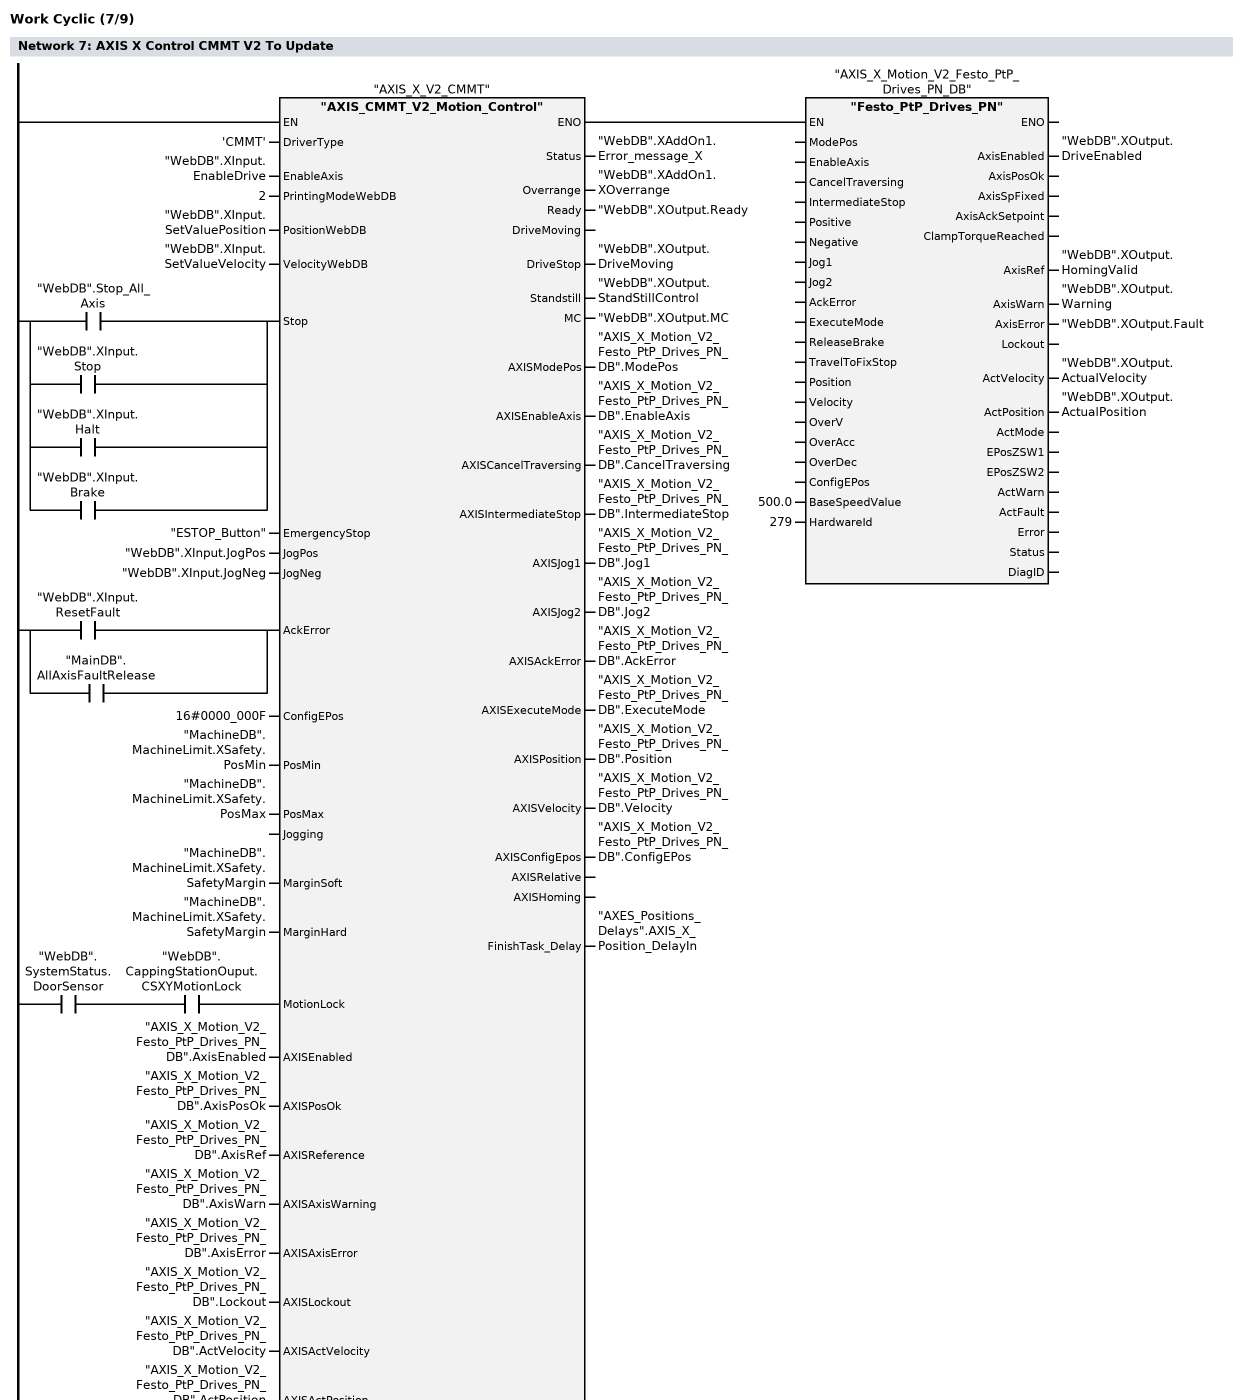
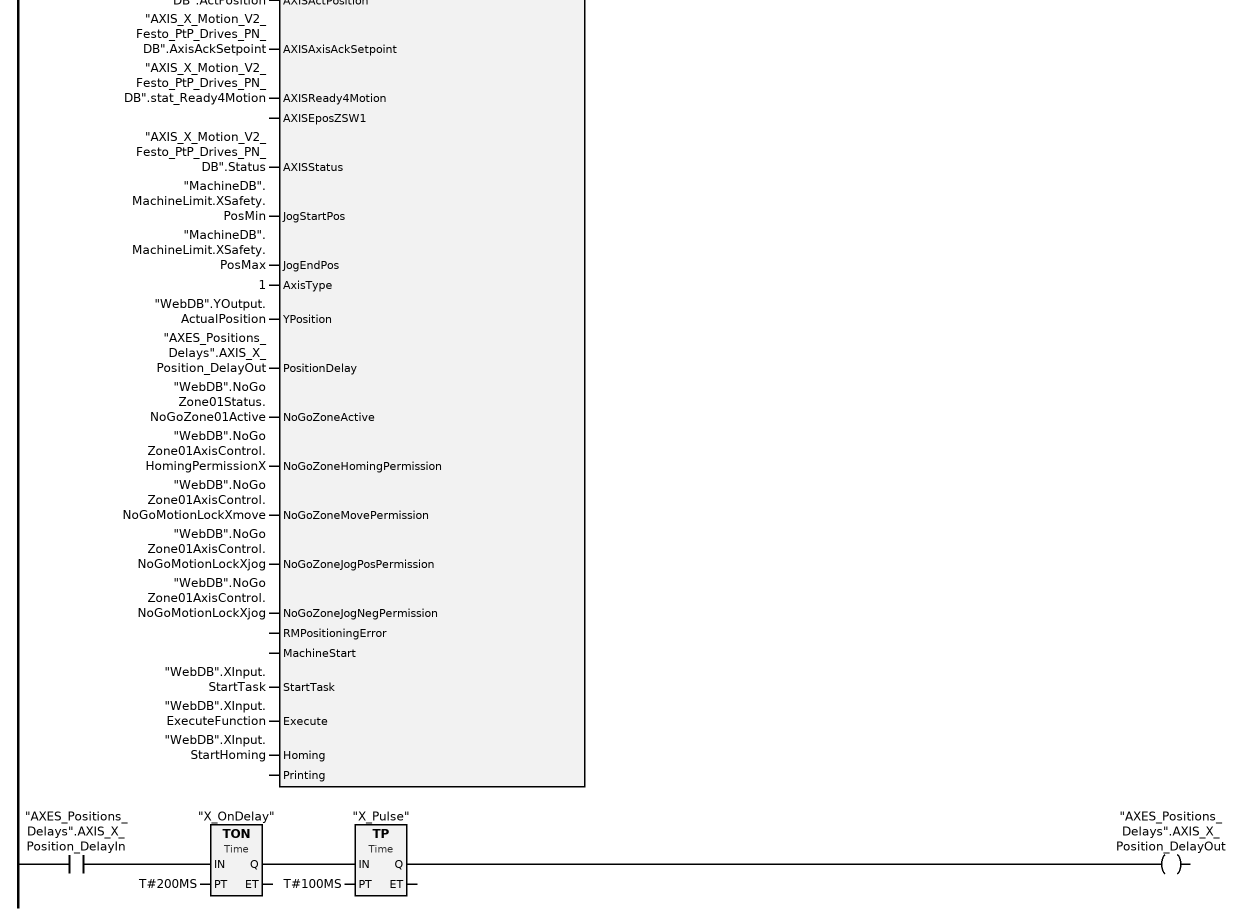
   RUNG wire#powerrail
      "AXIS_X_V2_CMMT"(Stop := wire#w1, AckError := wire#w2, MotionLock := wire#w3, DriverType := 'CMMT', EnableAxis := "WebDB".XInput.EnableDrive, PrintingModeWebDB := 2, PositionWebDB := "WebDB".XInput.SetValuePosition, VelocityWebDB := "WebDB".XInput.SetValueVelocity, EmergencyStop := "ESTOP_Button", JogPos := "WebDB".XInput.JogPos, JogNeg := "WebDB".XInput.JogNeg, ConfigEPos := 16#0000_000F, PosMin := "MachineDB".MachineLimit.XSafety.PosMin, PosMax := "MachineDB".MachineLimit.XSafety.PosMax, Jogging :=, MarginSoft := "MachineDB".MachineLimit.XSafety.SafetyMargin, MarginHard := "MachineDB".MachineLimit.XSafety.SafetyMargin, AXISEnabled := "AXIS_X_Motion_V2_Festo_PtP_Drives_PN_DB".AxisEnabled, AXISPosOk := "AXIS_X_Motion_V2_Festo_PtP_Drives_PN_DB".AxisPosOk, AXISReference := "AXIS_X_Motion_V2_Festo_PtP_Drives_PN_DB".AxisRef, AXISAxisWarning := "AXIS_X_Motion_V2_Festo_PtP_Drives_PN_DB".AxisWarn, AXISAxisError := "AXIS_X_Motion_V2_Festo_PtP_Drives_PN_DB".AxisError, AXISLockout := "AXIS_X_Motion_V2_Festo_PtP_Drives_PN_DB".Lockout, AXISActVelocity := "AXIS_X_Motion_V2_Festo_PtP_Drives_PN_DB".ActVelocity, AXISActPosition := "AXIS_X_Motion_V2_Festo_PtP_Drives_PN_DB".ActPosition, AXISAxisAckSetpoint := "AXIS_X_Motion_V2_Festo_PtP_Drives_PN_DB".AxisAckSetpoint, AXISReady4Motion := "AXIS_X_Motion_V2_Festo_PtP_Drives_PN_DB".stat_Ready4Motion, AXISEposZSW1 :=, AXISStatus := "AXIS_X_Motion_V2_Festo_PtP_Drives_PN_DB".Status, JogStartPos := "MachineDB".MachineLimit.XSafety.PosMin, JogEndPos := "MachineDB".MachineLimit.XSafety.PosMax, AxisType := 1, YPosition := "WebDB".YOutput.ActualPosition, PositionDelay := "AXES_Positions_Delays".AXIS_X_Position_DelayOut, NoGoZoneActive := "WebDB".NoGoZone01Status.NoGoZone01Active, NoGoZoneHomingPermission := "WebDB".NoGoZone01AxisControl.HomingPermissionX, NoGoZoneMovePermission := "WebDB".NoGoZone01AxisControl.NoGoMotionLockXmove, NoGoZoneJogPosPermission := "WebDB".NoGoZone01AxisControl.NoGoMotionLockXjog, NoGoZoneJogNegPermission := "WebDB".NoGoZone01AxisControl.NoGoMotionLockXjog, RMPositioningError :=, MachineStart :=, StartTask := "WebDB".XInput.StartTask, Execute := "WebDB".XInput.ExecuteFunction, Homing := "WebDB".XInput.StartHoming, Printing :=, Status => "WebDB".XAddOn1.Error_message_X, Overrange => "WebDB".XAddOn1.XOverrange, Ready => "WebDB".XOutput.Ready, DriveMoving =>, DriveStop => "WebDB".XOutput.DriveMoving, Standstill => "WebDB".XOutput.StandStillControl, MC => "WebDB".XOutput.MC, AXISModePos => "AXIS_X_Motion_V2_Festo_PtP_Drives_PN_DB".ModePos, AXISEnableAxis => "AXIS_X_Motion_V2_Festo_PtP_Drives_PN_DB".EnableAxis, AXISCancelTraversing => "AXIS_X_Motion_V2_Festo_PtP_Drives_PN_DB".CancelTraversing, AXISIntermediateStop => "AXIS_X_Motion_V2_Festo_PtP_Drives_PN_DB".IntermediateStop, AXISJog1 => "AXIS_X_Motion_V2_Festo_PtP_Drives_PN_DB".Jog1, AXISJog2 => "AXIS_X_Motion_V2_Festo_PtP_Drives_PN_DB".Jog2, AXISAckError => "AXIS_X_Motion_V2_Festo_PtP_Drives_PN_DB".AckError, AXISExecuteMode => "AXIS_X_Motion_V2_Festo_PtP_Drives_PN_DB".ExecuteMode, AXISPosition => "AXIS_X_Motion_V2_Festo_PtP_Drives_PN_DB".Position, AXISVelocity => "AXIS_X_Motion_V2_Festo_PtP_Drives_PN_DB".Velocity, AXISConfigEpos => "AXIS_X_Motion_V2_Festo_PtP_Drives_PN_DB".ConfigEPos, AXISRelative =>, AXISHoming =>, FinishTask_Delay => "AXES_Positions_Delays".AXIS_X_Position_DelayIn)
      "AXIS_X_Motion_V2_Festo_PtP_Drives_PN_DB"(ModePos :=, EnableAxis :=, CancelTraversing :=, IntermediateStop :=, Positive :=, Negative :=, Jog1 :=, Jog2 :=, AckError :=, ExecuteMode :=, ReleaseBrake :=, TravelToFixStop :=, Position :=, Velocity :=, OverV :=, OverAcc :=, OverDec :=, ConfigEPos :=, BaseSpeedValue := 500.0, HardwareId := 279, AxisEnabled => "WebDB".XOutput.DriveEnabled, AxisPosOk =>, AxisSpFixed =>, AxisAckSetpoint =>, ClampTorqueReached =>, AxisRef => "WebDB".XOutput.HomingValid, AxisWarn => "WebDB".XOutput.Warning, AxisError => "WebDB".XOutput.Fault, Lockout =>, ActVelocity => "WebDB".XOutput.ActualVelocity, ActPosition => "WebDB".XOutput.ActualPosition, ActMode =>, EPosZSW1 =>, EPosZSW2 =>, ActWarn =>, ActFault =>, Error =>, Status =>, DiagID =>)
   END_RUNG
   RUNG wire#powerrail
      Contact( "WebDB".Stop_All_Axis )
   END_RUNG wire#w1
   RUNG wire#powerrail
      Contact( "WebDB".XInput.Stop )
   END_RUNG wire#w1
   RUNG wire#powerrail
      Contact( "WebDB".XInput.Halt )
   END_RUNG wire#w1
   RUNG wire#powerrail
      Contact( "WebDB".XInput.Brake )
   END_RUNG wire#w1
   RUNG wire#powerrail
      Contact( "WebDB".XInput.ResetFault )
   END_RUNG wire#w2
   RUNG wire#powerrail
      Contact( "MainDB".AllAxisFaultRelease )
   END_RUNG wire#w2
   RUNG wire#powerrail
      Contact( "WebDB".SystemStatus.DoorSensor )
      Contact( "WebDB".CappingStationOuput.CSXYMotionLock )
   END_RUNG wire#w3
   RUNG wire#powerrail
      Contact( "AXES_Positions_Delays".AXIS_X_Position_DelayIn )
      { S7_Templates := "time_type := Time" } "X_OnDelay".TON(pt := T#200MS, et =>)
      { S7_Templates := "time_type := Time" } "X_Pulse".TP(pt := T#100MS, et =>)
      Coil( "AXES_Positions_Delays".AXIS_X_Position_DelayOut )
   END_RUNG
   // the same network as SCL:
   "AXIS_X_V2_CMMT"(DriverType := 'CMMT',   // "AXIS_CMMT_V2_Motion_Control"
                    EnableAxis := "WebDB".XInput.EnableDrive,
                    PrintingModeWebDB := 2,
                    PositionWebDB := "WebDB".XInput.SetValuePosition,
                    VelocityWebDB := "WebDB".XInput.SetValueVelocity,
                    Stop := "WebDB".Stop_All_Axis OR "WebDB".XInput.Stop OR "WebDB".XInput.Halt OR "WebDB".XInput.Brake,
                    EmergencyStop := "ESTOP_Button",
                    JogPos := "WebDB".XInput.JogPos,
                    JogNeg := "WebDB".XInput.JogNeg,
                    AckError := "WebDB".XInput.ResetFault OR "MainDB".AllAxisFaultRelease,
                    ConfigEPos := 16#0000_000F,
                    PosMin := "MachineDB".MachineLimit.XSafety.PosMin,
                    PosMax := "MachineDB".MachineLimit.XSafety.PosMax,
                    MarginSoft := "MachineDB".MachineLimit.XSafety.SafetyMargin,
                    MarginHard := "MachineDB".MachineLimit.XSafety.SafetyMargin,
                    MotionLock := "WebDB".SystemStatus.DoorSensor AND "WebDB".CappingStationOuput.CSXYMotionLock,
                    AXISEnabled := "AXIS_X_Motion_V2_Festo_PtP_Drives_PN_DB".AxisEnabled,
                    AXISPosOk := "AXIS_X_Motion_V2_Festo_PtP_Drives_PN_DB".AxisPosOk,
                    AXISReference := "AXIS_X_Motion_V2_Festo_PtP_Drives_PN_DB".AxisRef,
                    AXISAxisWarning := "AXIS_X_Motion_V2_Festo_PtP_Drives_PN_DB".AxisWarn,
                    AXISAxisError := "AXIS_X_Motion_V2_Festo_PtP_Drives_PN_DB".AxisError,
                    AXISLockout := "AXIS_X_Motion_V2_Festo_PtP_Drives_PN_DB".Lockout,
                    AXISActVelocity := "AXIS_X_Motion_V2_Festo_PtP_Drives_PN_DB".ActVelocity,
                    AXISActPosition := "AXIS_X_Motion_V2_Festo_PtP_Drives_PN_DB".ActPosition,
                    AXISAxisAckSetpoint := "AXIS_X_Motion_V2_Festo_PtP_Drives_PN_DB".AxisAckSetpoint,
                    AXISReady4Motion := "AXIS_X_Motion_V2_Festo_PtP_Drives_PN_DB".stat_Ready4Motion,
                    AXISStatus := "AXIS_X_Motion_V2_Festo_PtP_Drives_PN_DB".Status,
                    JogStartPos := "MachineDB".MachineLimit.XSafety.PosMin,
                    JogEndPos := "MachineDB".MachineLimit.XSafety.PosMax,
                    AxisType := 1,
                    YPosition := "WebDB".YOutput.ActualPosition,
                    PositionDelay := "AXES_Positions_Delays".AXIS_X_Position_DelayOut,
                    NoGoZoneActive := "WebDB".NoGoZone01Status.NoGoZone01Active,
                    NoGoZoneHomingPermission := "WebDB".NoGoZone01AxisControl.HomingPermissionX,
                    NoGoZoneMovePermission := "WebDB".NoGoZone01AxisControl.NoGoMotionLockXmove,
                    NoGoZoneJogPosPermission := "WebDB".NoGoZone01AxisControl.NoGoMotionLockXjog,
                    NoGoZoneJogNegPermission := "WebDB".NoGoZone01AxisControl.NoGoMotionLockXjog,
                    StartTask := "WebDB".XInput.StartTask,
                    Execute := "WebDB".XInput.ExecuteFunction,
                    Homing := "WebDB".XInput.StartHoming,
                    Status => "WebDB".XAddOn1.Error_message_X,
                    Overrange => "WebDB".XAddOn1.XOverrange,
                    Ready => "WebDB".XOutput.Ready,
                    DriveStop => "WebDB".XOutput.DriveMoving,
                    Standstill => "WebDB".XOutput.StandStillControl,
                    MC => "WebDB".XOutput.MC,
                    AXISModePos => "AXIS_X_Motion_V2_Festo_PtP_Drives_PN_DB".ModePos,
                    AXISEnableAxis => "AXIS_X_Motion_V2_Festo_PtP_Drives_PN_DB".EnableAxis,
                    AXISCancelTraversing => "AXIS_X_Motion_V2_Festo_PtP_Drives_PN_DB".CancelTraversing,
                    AXISIntermediateStop => "AXIS_X_Motion_V2_Festo_PtP_Drives_PN_DB".IntermediateStop,
                    AXISJog1 => "AXIS_X_Motion_V2_Festo_PtP_Drives_PN_DB".Jog1,
                    AXISJog2 => "AXIS_X_Motion_V2_Festo_PtP_Drives_PN_DB".Jog2,
                    AXISAckError => "AXIS_X_Motion_V2_Festo_PtP_Drives_PN_DB".AckError,
                    AXISExecuteMode => "AXIS_X_Motion_V2_Festo_PtP_Drives_PN_DB".ExecuteMode,
                    AXISPosition => "AXIS_X_Motion_V2_Festo_PtP_Drives_PN_DB".Position,
                    AXISVelocity => "AXIS_X_Motion_V2_Festo_PtP_Drives_PN_DB".Velocity,
                    AXISConfigEpos => "AXIS_X_Motion_V2_Festo_PtP_Drives_PN_DB".ConfigEPos,
                    FinishTask_Delay => "AXES_Positions_Delays".AXIS_X_Position_DelayIn,
                    ENO => #_w1);
   IF #_w1 THEN
       "AXIS_X_Motion_V2_Festo_PtP_Drives_PN_DB"(BaseSpeedValue := 500.0,   // "Festo_PtP_Drives_PN"
                               HardwareId := 279,
                               AxisEnabled => "WebDB".XOutput.DriveEnabled,
                               AxisRef => "WebDB".XOutput.HomingValid,
                               AxisWarn => "WebDB".XOutput.Warning,
                               AxisError => "WebDB".XOutput.Fault,
                               ActVelocity => "WebDB".XOutput.ActualVelocity,
                               ActPosition => "WebDB".XOutput.ActualPosition);
   END_IF;
   "X_OnDelay".TON(IN := "AXES_Positions_Delays".AXIS_X_Position_DelayIn, PT := T#200MS);
   "X_Pulse".TP(IN := "X_OnDelay".Q, PT := T#100MS);
   "AXES_Positions_Delays".AXIS_X_Position_DelayOut := "X_Pulse".Q;
END_REGION

REGION Network 8: AXIS Y Control CMMT V2 To Update
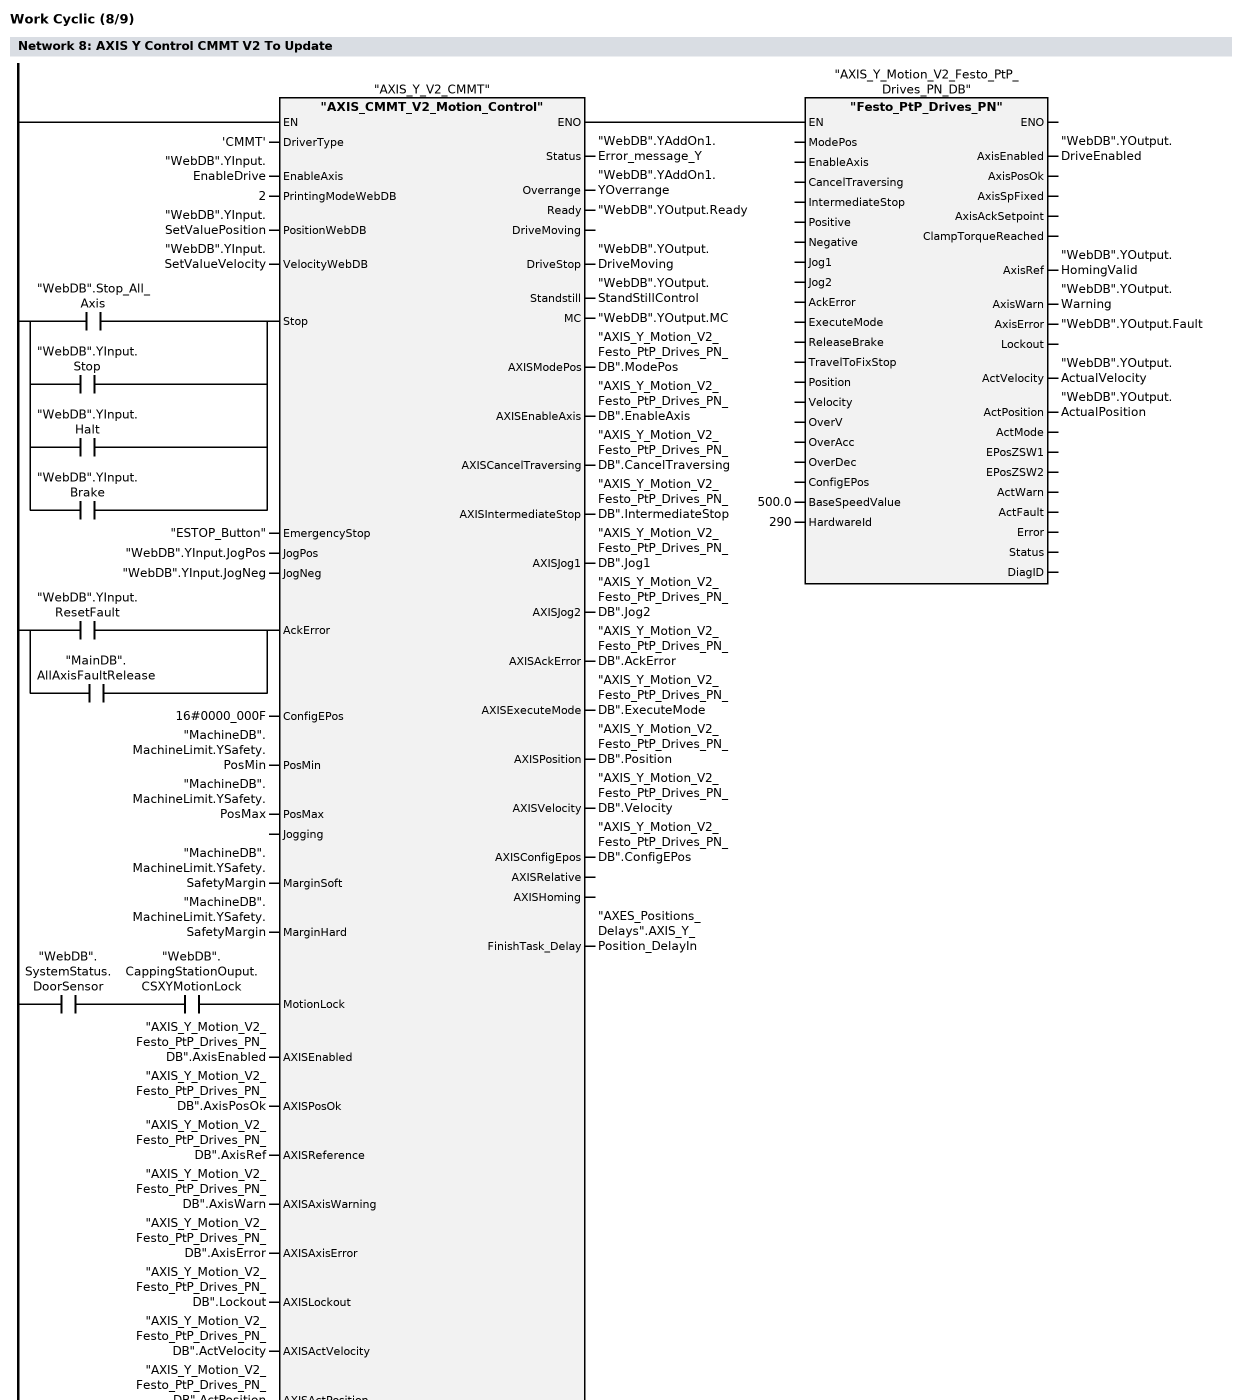
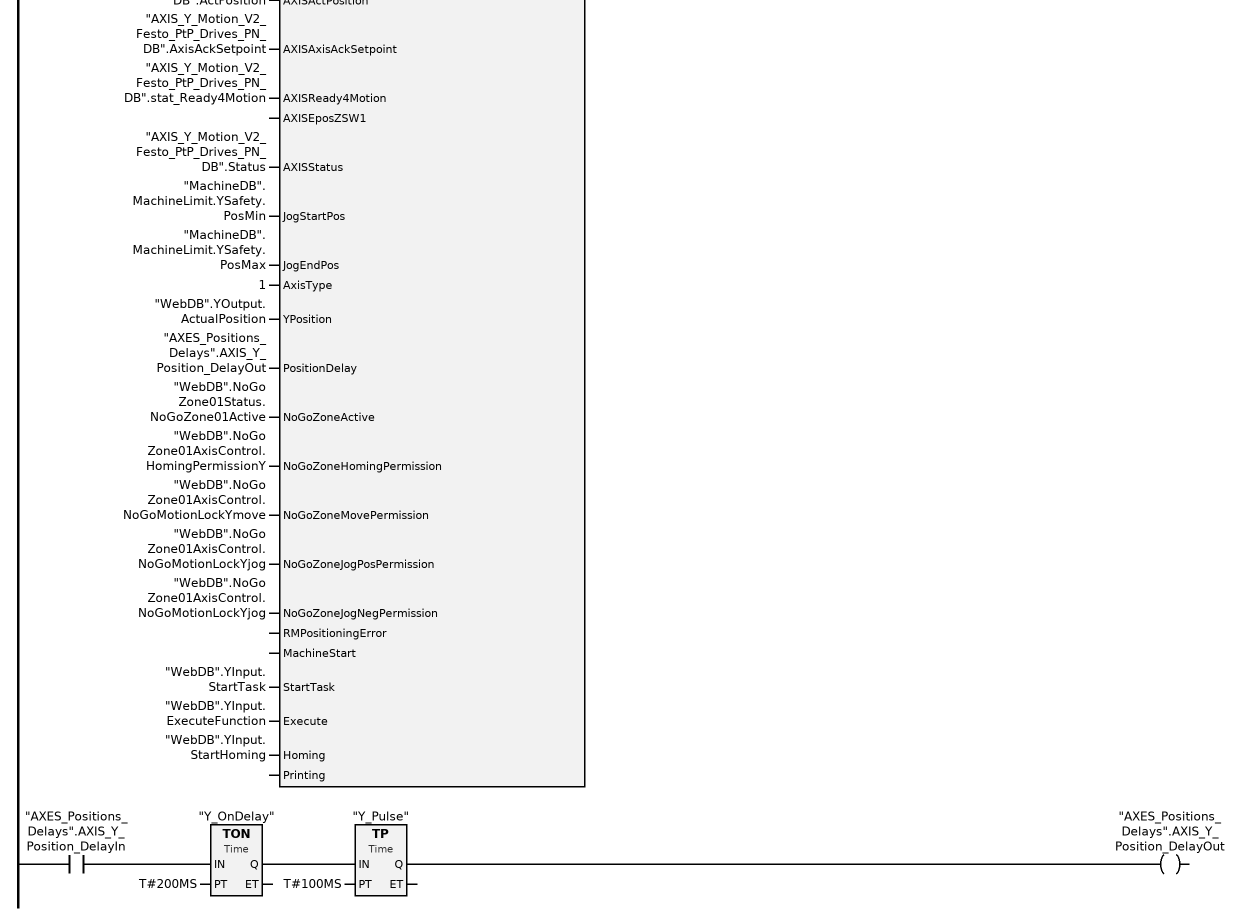
   RUNG wire#powerrail
      "AXIS_Y_V2_CMMT"(Stop := wire#w1, AckError := wire#w2, MotionLock := wire#w3, DriverType := 'CMMT', EnableAxis := "WebDB".YInput.EnableDrive, PrintingModeWebDB := 2, PositionWebDB := "WebDB".YInput.SetValuePosition, VelocityWebDB := "WebDB".YInput.SetValueVelocity, EmergencyStop := "ESTOP_Button", JogPos := "WebDB".YInput.JogPos, JogNeg := "WebDB".YInput.JogNeg, ConfigEPos := 16#0000_000F, PosMin := "MachineDB".MachineLimit.YSafety.PosMin, PosMax := "MachineDB".MachineLimit.YSafety.PosMax, Jogging :=, MarginSoft := "MachineDB".MachineLimit.YSafety.SafetyMargin, MarginHard := "MachineDB".MachineLimit.YSafety.SafetyMargin, AXISEnabled := "AXIS_Y_Motion_V2_Festo_PtP_Drives_PN_DB".AxisEnabled, AXISPosOk := "AXIS_Y_Motion_V2_Festo_PtP_Drives_PN_DB".AxisPosOk, AXISReference := "AXIS_Y_Motion_V2_Festo_PtP_Drives_PN_DB".AxisRef, AXISAxisWarning := "AXIS_Y_Motion_V2_Festo_PtP_Drives_PN_DB".AxisWarn, AXISAxisError := "AXIS_Y_Motion_V2_Festo_PtP_Drives_PN_DB".AxisError, AXISLockout := "AXIS_Y_Motion_V2_Festo_PtP_Drives_PN_DB".Lockout, AXISActVelocity := "AXIS_Y_Motion_V2_Festo_PtP_Drives_PN_DB".ActVelocity, AXISActPosition := "AXIS_Y_Motion_V2_Festo_PtP_Drives_PN_DB".ActPosition, AXISAxisAckSetpoint := "AXIS_Y_Motion_V2_Festo_PtP_Drives_PN_DB".AxisAckSetpoint, AXISReady4Motion := "AXIS_Y_Motion_V2_Festo_PtP_Drives_PN_DB".stat_Ready4Motion, AXISEposZSW1 :=, AXISStatus := "AXIS_Y_Motion_V2_Festo_PtP_Drives_PN_DB".Status, JogStartPos := "MachineDB".MachineLimit.YSafety.PosMin, JogEndPos := "MachineDB".MachineLimit.YSafety.PosMax, AxisType := 1, YPosition := "WebDB".YOutput.ActualPosition, PositionDelay := "AXES_Positions_Delays".AXIS_Y_Position_DelayOut, NoGoZoneActive := "WebDB".NoGoZone01Status.NoGoZone01Active, NoGoZoneHomingPermission := "WebDB".NoGoZone01AxisControl.HomingPermissionY, NoGoZoneMovePermission := "WebDB".NoGoZone01AxisControl.NoGoMotionLockYmove, NoGoZoneJogPosPermission := "WebDB".NoGoZone01AxisControl.NoGoMotionLockYjog, NoGoZoneJogNegPermission := "WebDB".NoGoZone01AxisControl.NoGoMotionLockYjog, RMPositioningError :=, MachineStart :=, StartTask := "WebDB".YInput.StartTask, Execute := "WebDB".YInput.ExecuteFunction, Homing := "WebDB".YInput.StartHoming, Printing :=, Status => "WebDB".YAddOn1.Error_message_Y, Overrange => "WebDB".YAddOn1.YOverrange, Ready => "WebDB".YOutput.Ready, DriveMoving =>, DriveStop => "WebDB".YOutput.DriveMoving, Standstill => "WebDB".YOutput.StandStillControl, MC => "WebDB".YOutput.MC, AXISModePos => "AXIS_Y_Motion_V2_Festo_PtP_Drives_PN_DB".ModePos, AXISEnableAxis => "AXIS_Y_Motion_V2_Festo_PtP_Drives_PN_DB".EnableAxis, AXISCancelTraversing => "AXIS_Y_Motion_V2_Festo_PtP_Drives_PN_DB".CancelTraversing, AXISIntermediateStop => "AXIS_Y_Motion_V2_Festo_PtP_Drives_PN_DB".IntermediateStop, AXISJog1 => "AXIS_Y_Motion_V2_Festo_PtP_Drives_PN_DB".Jog1, AXISJog2 => "AXIS_Y_Motion_V2_Festo_PtP_Drives_PN_DB".Jog2, AXISAckError => "AXIS_Y_Motion_V2_Festo_PtP_Drives_PN_DB".AckError, AXISExecuteMode => "AXIS_Y_Motion_V2_Festo_PtP_Drives_PN_DB".ExecuteMode, AXISPosition => "AXIS_Y_Motion_V2_Festo_PtP_Drives_PN_DB".Position, AXISVelocity => "AXIS_Y_Motion_V2_Festo_PtP_Drives_PN_DB".Velocity, AXISConfigEpos => "AXIS_Y_Motion_V2_Festo_PtP_Drives_PN_DB".ConfigEPos, AXISRelative =>, AXISHoming =>, FinishTask_Delay => "AXES_Positions_Delays".AXIS_Y_Position_DelayIn)
      "AXIS_Y_Motion_V2_Festo_PtP_Drives_PN_DB"(ModePos :=, EnableAxis :=, CancelTraversing :=, IntermediateStop :=, Positive :=, Negative :=, Jog1 :=, Jog2 :=, AckError :=, ExecuteMode :=, ReleaseBrake :=, TravelToFixStop :=, Position :=, Velocity :=, OverV :=, OverAcc :=, OverDec :=, ConfigEPos :=, BaseSpeedValue := 500.0, HardwareId := 290, AxisEnabled => "WebDB".YOutput.DriveEnabled, AxisPosOk =>, AxisSpFixed =>, AxisAckSetpoint =>, ClampTorqueReached =>, AxisRef => "WebDB".YOutput.HomingValid, AxisWarn => "WebDB".YOutput.Warning, AxisError => "WebDB".YOutput.Fault, Lockout =>, ActVelocity => "WebDB".YOutput.ActualVelocity, ActPosition => "WebDB".YOutput.ActualPosition, ActMode =>, EPosZSW1 =>, EPosZSW2 =>, ActWarn =>, ActFault =>, Error =>, Status =>, DiagID =>)
   END_RUNG
   RUNG wire#powerrail
      Contact( "WebDB".Stop_All_Axis )
   END_RUNG wire#w1
   RUNG wire#powerrail
      Contact( "WebDB".YInput.Stop )
   END_RUNG wire#w1
   RUNG wire#powerrail
      Contact( "WebDB".YInput.Halt )
   END_RUNG wire#w1
   RUNG wire#powerrail
      Contact( "WebDB".YInput.Brake )
   END_RUNG wire#w1
   RUNG wire#powerrail
      Contact( "WebDB".YInput.ResetFault )
   END_RUNG wire#w2
   RUNG wire#powerrail
      Contact( "MainDB".AllAxisFaultRelease )
   END_RUNG wire#w2
   RUNG wire#powerrail
      Contact( "WebDB".SystemStatus.DoorSensor )
      Contact( "WebDB".CappingStationOuput.CSXYMotionLock )
   END_RUNG wire#w3
   RUNG wire#powerrail
      Contact( "AXES_Positions_Delays".AXIS_Y_Position_DelayIn )
      { S7_Templates := "time_type := Time" } "Y_OnDelay".TON(pt := T#200MS, et =>)
      { S7_Templates := "time_type := Time" } "Y_Pulse".TP(pt := T#100MS, et =>)
      Coil( "AXES_Positions_Delays".AXIS_Y_Position_DelayOut )
   END_RUNG
   // the same network as SCL:
   "AXIS_Y_V2_CMMT"(DriverType := 'CMMT',   // "AXIS_CMMT_V2_Motion_Control"
                    EnableAxis := "WebDB".YInput.EnableDrive,
                    PrintingModeWebDB := 2,
                    PositionWebDB := "WebDB".YInput.SetValuePosition,
                    VelocityWebDB := "WebDB".YInput.SetValueVelocity,
                    Stop := "WebDB".Stop_All_Axis OR "WebDB".YInput.Stop OR "WebDB".YInput.Halt OR "WebDB".YInput.Brake,
                    EmergencyStop := "ESTOP_Button",
                    JogPos := "WebDB".YInput.JogPos,
                    JogNeg := "WebDB".YInput.JogNeg,
                    AckError := "WebDB".YInput.ResetFault OR "MainDB".AllAxisFaultRelease,
                    ConfigEPos := 16#0000_000F,
                    PosMin := "MachineDB".MachineLimit.YSafety.PosMin,
                    PosMax := "MachineDB".MachineLimit.YSafety.PosMax,
                    MarginSoft := "MachineDB".MachineLimit.YSafety.SafetyMargin,
                    MarginHard := "MachineDB".MachineLimit.YSafety.SafetyMargin,
                    MotionLock := "WebDB".SystemStatus.DoorSensor AND "WebDB".CappingStationOuput.CSXYMotionLock,
                    AXISEnabled := "AXIS_Y_Motion_V2_Festo_PtP_Drives_PN_DB".AxisEnabled,
                    AXISPosOk := "AXIS_Y_Motion_V2_Festo_PtP_Drives_PN_DB".AxisPosOk,
                    AXISReference := "AXIS_Y_Motion_V2_Festo_PtP_Drives_PN_DB".AxisRef,
                    AXISAxisWarning := "AXIS_Y_Motion_V2_Festo_PtP_Drives_PN_DB".AxisWarn,
                    AXISAxisError := "AXIS_Y_Motion_V2_Festo_PtP_Drives_PN_DB".AxisError,
                    AXISLockout := "AXIS_Y_Motion_V2_Festo_PtP_Drives_PN_DB".Lockout,
                    AXISActVelocity := "AXIS_Y_Motion_V2_Festo_PtP_Drives_PN_DB".ActVelocity,
                    AXISActPosition := "AXIS_Y_Motion_V2_Festo_PtP_Drives_PN_DB".ActPosition,
                    AXISAxisAckSetpoint := "AXIS_Y_Motion_V2_Festo_PtP_Drives_PN_DB".AxisAckSetpoint,
                    AXISReady4Motion := "AXIS_Y_Motion_V2_Festo_PtP_Drives_PN_DB".stat_Ready4Motion,
                    AXISStatus := "AXIS_Y_Motion_V2_Festo_PtP_Drives_PN_DB".Status,
                    JogStartPos := "MachineDB".MachineLimit.YSafety.PosMin,
                    JogEndPos := "MachineDB".MachineLimit.YSafety.PosMax,
                    AxisType := 1,
                    YPosition := "WebDB".YOutput.ActualPosition,
                    PositionDelay := "AXES_Positions_Delays".AXIS_Y_Position_DelayOut,
                    NoGoZoneActive := "WebDB".NoGoZone01Status.NoGoZone01Active,
                    NoGoZoneHomingPermission := "WebDB".NoGoZone01AxisControl.HomingPermissionY,
                    NoGoZoneMovePermission := "WebDB".NoGoZone01AxisControl.NoGoMotionLockYmove,
                    NoGoZoneJogPosPermission := "WebDB".NoGoZone01AxisControl.NoGoMotionLockYjog,
                    NoGoZoneJogNegPermission := "WebDB".NoGoZone01AxisControl.NoGoMotionLockYjog,
                    StartTask := "WebDB".YInput.StartTask,
                    Execute := "WebDB".YInput.ExecuteFunction,
                    Homing := "WebDB".YInput.StartHoming,
                    Status => "WebDB".YAddOn1.Error_message_Y,
                    Overrange => "WebDB".YAddOn1.YOverrange,
                    Ready => "WebDB".YOutput.Ready,
                    DriveStop => "WebDB".YOutput.DriveMoving,
                    Standstill => "WebDB".YOutput.StandStillControl,
                    MC => "WebDB".YOutput.MC,
                    AXISModePos => "AXIS_Y_Motion_V2_Festo_PtP_Drives_PN_DB".ModePos,
                    AXISEnableAxis => "AXIS_Y_Motion_V2_Festo_PtP_Drives_PN_DB".EnableAxis,
                    AXISCancelTraversing => "AXIS_Y_Motion_V2_Festo_PtP_Drives_PN_DB".CancelTraversing,
                    AXISIntermediateStop => "AXIS_Y_Motion_V2_Festo_PtP_Drives_PN_DB".IntermediateStop,
                    AXISJog1 => "AXIS_Y_Motion_V2_Festo_PtP_Drives_PN_DB".Jog1,
                    AXISJog2 => "AXIS_Y_Motion_V2_Festo_PtP_Drives_PN_DB".Jog2,
                    AXISAckError => "AXIS_Y_Motion_V2_Festo_PtP_Drives_PN_DB".AckError,
                    AXISExecuteMode => "AXIS_Y_Motion_V2_Festo_PtP_Drives_PN_DB".ExecuteMode,
                    AXISPosition => "AXIS_Y_Motion_V2_Festo_PtP_Drives_PN_DB".Position,
                    AXISVelocity => "AXIS_Y_Motion_V2_Festo_PtP_Drives_PN_DB".Velocity,
                    AXISConfigEpos => "AXIS_Y_Motion_V2_Festo_PtP_Drives_PN_DB".ConfigEPos,
                    FinishTask_Delay => "AXES_Positions_Delays".AXIS_Y_Position_DelayIn,
                    ENO => #_w1);
   IF #_w1 THEN
       "AXIS_Y_Motion_V2_Festo_PtP_Drives_PN_DB"(BaseSpeedValue := 500.0,   // "Festo_PtP_Drives_PN"
                               HardwareId := 290,
                               AxisEnabled => "WebDB".YOutput.DriveEnabled,
                               AxisRef => "WebDB".YOutput.HomingValid,
                               AxisWarn => "WebDB".YOutput.Warning,
                               AxisError => "WebDB".YOutput.Fault,
                               ActVelocity => "WebDB".YOutput.ActualVelocity,
                               ActPosition => "WebDB".YOutput.ActualPosition);
   END_IF;
   "Y_OnDelay".TON(IN := "AXES_Positions_Delays".AXIS_Y_Position_DelayIn, PT := T#200MS);
   "Y_Pulse".TP(IN := "Y_OnDelay".Q, PT := T#100MS);
   "AXES_Positions_Delays".AXIS_Y_Position_DelayOut := "Y_Pulse".Q;
END_REGION

REGION Network 9: Roller V3
   // The RollerV3 block already writes the roller speed and direction to the technology object. This means that the outputs are no longer needed.
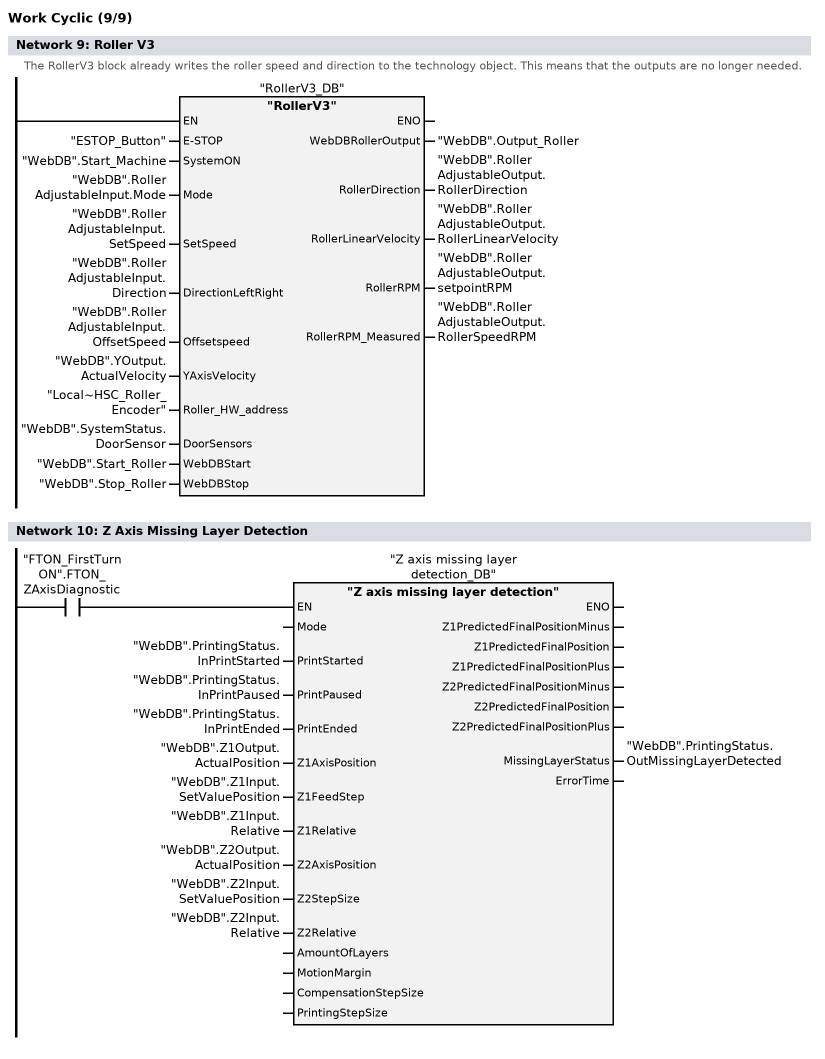
   RUNG wire#powerrail
      "RollerV3_DB"("E-STOP" := "ESTOP_Button", SystemON := "WebDB".Start_Machine, Mode := "WebDB".RollerAdjustableInput.Mode, SetSpeed := "WebDB".RollerAdjustableInput.SetSpeed, DirectionLeftRight := "WebDB".RollerAdjustableInput.Direction, Offsetspeed := "WebDB".RollerAdjustableInput.OffsetSpeed, YAxisVelocity := "WebDB".YOutput.ActualVelocity, Roller_HW_address := "Local~HSC_Roller_Encoder", DoorSensors := "WebDB".SystemStatus.DoorSensor, WebDBStart := "WebDB".Start_Roller, WebDBStop := "WebDB".Stop_Roller, WebDBRollerOutput => "WebDB".Output_Roller, RollerDirection => "WebDB".RollerAdjustableOutput.RollerDirection, RollerLinearVelocity => "WebDB".RollerAdjustableOutput.RollerLinearVelocity, RollerRPM => "WebDB".RollerAdjustableOutput.setpointRPM, RollerRPM_Measured => "WebDB".RollerAdjustableOutput.RollerSpeedRPM)
   END_RUNG
   // the same network as SCL:
   "RollerV3_DB"("E-STOP" := "ESTOP_Button",   // "RollerV3"
                 SystemON := "WebDB".Start_Machine,
                 Mode := "WebDB".RollerAdjustableInput.Mode,
                 SetSpeed := "WebDB".RollerAdjustableInput.SetSpeed,
                 DirectionLeftRight := "WebDB".RollerAdjustableInput.Direction,
                 Offsetspeed := "WebDB".RollerAdjustableInput.OffsetSpeed,
                 YAxisVelocity := "WebDB".YOutput.ActualVelocity,
                 Roller_HW_address := "Local~HSC_Roller_Encoder",
                 DoorSensors := "WebDB".SystemStatus.DoorSensor,
                 WebDBStart := "WebDB".Start_Roller,
                 WebDBStop := "WebDB".Stop_Roller,
                 WebDBRollerOutput => "WebDB".Output_Roller,
                 RollerDirection => "WebDB".RollerAdjustableOutput.RollerDirection,
                 RollerLinearVelocity => "WebDB".RollerAdjustableOutput.RollerLinearVelocity,
                 RollerRPM => "WebDB".RollerAdjustableOutput.setpointRPM,
                 RollerRPM_Measured => "WebDB".RollerAdjustableOutput.RollerSpeedRPM);
END_REGION

REGION Network 10: Z Axis Missing Layer Detection
   RUNG wire#powerrail
      Contact( "FTON_FirstTurnON".FTON_ZAxisDiagnostic )
      "Z axis missing layer detection_DB"(Mode :=, PrintStarted := "WebDB".PrintingStatus.InPrintStarted, PrintPaused := "WebDB".PrintingStatus.InPrintPaused, PrintEnded := "WebDB".PrintingStatus.InPrintEnded, Z1AxisPosition := "WebDB".Z1Output.ActualPosition, Z1FeedStep := "WebDB".Z1Input.SetValuePosition, Z1Relative := "WebDB".Z1Input.Relative, Z2AxisPosition := "WebDB".Z2Output.ActualPosition, Z2StepSize := "WebDB".Z2Input.SetValuePosition, Z2Relative := "WebDB".Z2Input.Relative, AmountOfLayers :=, MotionMargin :=, CompensationStepSize :=, PrintingStepSize :=, Z1PredictedFinalPositionMinus =>, Z1PredictedFinalPosition =>, Z1PredictedFinalPositionPlus =>, Z2PredictedFinalPositionMinus =>, Z2PredictedFinalPosition =>, Z2PredictedFinalPositionPlus =>, MissingLayerStatus => "WebDB".PrintingStatus.OutMissingLayerDetected, ErrorTime =>)
   END_RUNG
   // the same network as SCL:
   IF "FTON_FirstTurnON".FTON_ZAxisDiagnostic THEN
       "Z axis missing layer detection_DB"(PrintStarted := "WebDB".PrintingStatus.InPrintStarted,   // "Z axis missing layer detection"
                               PrintPaused := "WebDB".PrintingStatus.InPrintPaused,
                               PrintEnded := "WebDB".PrintingStatus.InPrintEnded,
                               Z1AxisPosition := "WebDB".Z1Output.ActualPosition,
                               Z1FeedStep := "WebDB".Z1Input.SetValuePosition,
                               Z1Relative := "WebDB".Z1Input.Relative,
                               Z2AxisPosition := "WebDB".Z2Output.ActualPosition,
                               Z2StepSize := "WebDB".Z2Input.SetValuePosition,
                               Z2Relative := "WebDB".Z2Input.Relative,
                               MissingLayerStatus => "WebDB".PrintingStatus.OutMissingLayerDetected);
   END_IF;
END_REGION
END_ORGANIZATION_BLOCK

FUNCTION_BLOCK "AXIS_CMMT_V2_Motion_Control"   // FB22, LAD
TITLE = Description
{ S7_Optimized_Access := 'TRUE' }
VERSION : 0.1
// This is the motion function block used to control all the axes. Due to some differences in the control part for different types of motion and drives, there are additional conditions in some parts of the code.
// 
// Important things to check if the drive is not moving:
// - homing
// - motion lock from add ons (capping station, no go zones)
// - door sensors
// - operation mode
// - communication with the drives (Online access)
   VAR_INPUT
      DriverType : String;   // CMMT; CMMS;
      EnableAxis : Bool;
      PrintingModeWebDB : Int;   // Used while executing the movement
      PositionWebDB : DInt;
      VelocityWebDB : Real;
      Stop : Bool;
      EmergencyStop : Bool;
      JogPos : Bool;
      JogNeg : Bool;
      AckError : Bool;
      ConfigEPos : DWord;
      PosMin : DInt;
      PosMax : DInt;
      Jogging : Bool;
      MarginSoft : DInt;
      MarginHard : DInt;
      MotionLock : Bool;   // Axis will not move is this bool is 0
      AXISEnabled : Bool;
      AXISPosOk : Bool;
      AXISReference : Bool;
      AXISAxisWarning : Bool;
      AXISAxisError : Bool;
      AXISLockout : Bool;
      AXISActVelocity : Real;
      AXISActPosition : DInt;
      AXISAxisAckSetpoint : Bool;
      AXISReady4Motion : Bool;
      AXISEposZSW1 : Word;
      AXISStatus : Word;
      JogStartPos : DInt;   // Limit for jogging
      JogEndPos : DInt;   // Limit for jogging
      AxisType : Int;   // Axis Type: 1 - X; 2 - Y; 3 - Z1; 4 - Z2
      YPosition : DInt;
      PositionDelay : Bool;   // Delay to make it easier to confirm that the motion was finished
      NoGoZoneActive : Bool;   // 1 to activate no go zone
      NoGoZoneHomingPermission : Bool;
      NoGoZoneMovePermission : Bool;
      NoGoZoneJogPosPermission : Bool;
      NoGoZoneJogNegPermission : Bool;
      RMPositioningError : DInt := 5;   // Input Relativer Motion Position Error that we accept
      MachineStart : Bool;
   END_VAR
   VAR_OUTPUT
      Status : Word;
      Overrange : Bool;
      Ready : Bool;
      DriveMoving : Bool;
      DriveStop : Bool;
      Standstill : Bool;
      MC : Bool;
      AXISModePos : Int;
      AXISEnableAxis : Bool;
      AXISCancelTraversing : Bool;
      AXISIntermediateStop : Bool;
      AXISJog1 : Bool;
      AXISJog2 : Bool;
      AXISAckError : Bool;
      AXISExecuteMode : Bool;
      AXISPosition : DInt;
      AXISVelocity : Real;
      AXISConfigEpos : DWord;
      AXISRelative : Bool;
      AXISHoming : Bool;
      FinishTask_Delay : Bool;
   END_VAR
   VAR_IN_OUT
      StartTask : Bool;
      Execute : Bool;
      Homing : Bool;
      Printing : Bool;
   END_VAR
   VAR
      ExecutingMemory : Bool;
      HomingMemory : Bool;
      TaskMemory : Bool;
      ModePos : Int := 4;
      PosOk : Bool;
      Reference : Bool;
      PositionInternal : DInt;
      LockoutInternal : Bool;
      RelativeMode : Bool;   // Mode 1
      AbsoluteMode : Bool;   // Mode 2
      TaskFinished : Bool;
      JoggingXPermission : Bool;
      JoggingYPermission : Bool;
      JoggingPOSZ1Z2Permission : Bool;
      JoggingNEGZ1Z2Permission : Bool;
      JoggingPosMax : DInt;
      JoggingPosMin : DInt;
      JoggingPositionCorrection : DInt := 1500;
      ProfinetDisconnected : Bool;
      PositionStepPlus : DInt;
      CMMT : Bool;
      CMMS : Bool;
      RMStepStartPosition : DInt;   // Relative Motion Step Start Position
      RMPredictedPosition : DInt;   // Relative Motion Predicted Position
      RMFinalPosition : DInt;   // Relative Motion Final Position
      RMLastStepPositionError : DInt;   // Relative Motion Last Step Position Error
      RMStartTaskM01 : Bool;   // Relative Motion Start Task M Positive
      RMStartTaksM02 : Bool;   // Relative Motion Start Task M Negative
      RMStepRangePlus : DInt;
      RMStepRangeMinus : DInt;
      RelativeDirectionInRange : Bool;
   END_VAR
   VAR_TEMP
      RelativeModeHomingM : Bool;
      Jog1_pos : Bool;   // Jog positive direction
      Jog2_neg : Bool;   // Jog negative direction
      Memory1 : Bool;
      Memory2 : Bool;
      PosMinSoft : DInt;
      PosMaxSoft : DInt;
      InternalError : Bool;
      InternalWarning : Bool;
      ExecuteBusy : Bool;
      ExecutingInternal : Bool;
      HomingInternal : Bool;
      TaskInternal : Bool;
      Position_Plus : DInt;
      Position_Minus : DInt;
      TestFinished : Bool;
   END_VAR
   VAR CONSTANT
      Position_Error : DInt := 10;
   END_VAR
   VAR_TEMP   // added for the SCL form of the ladder/FBD networks
      _w1 : Bool;
      _w2 : Bool;
      _w3 : Bool;
   END_VAR
BEGIN

REGION Network 1: Checking driver type
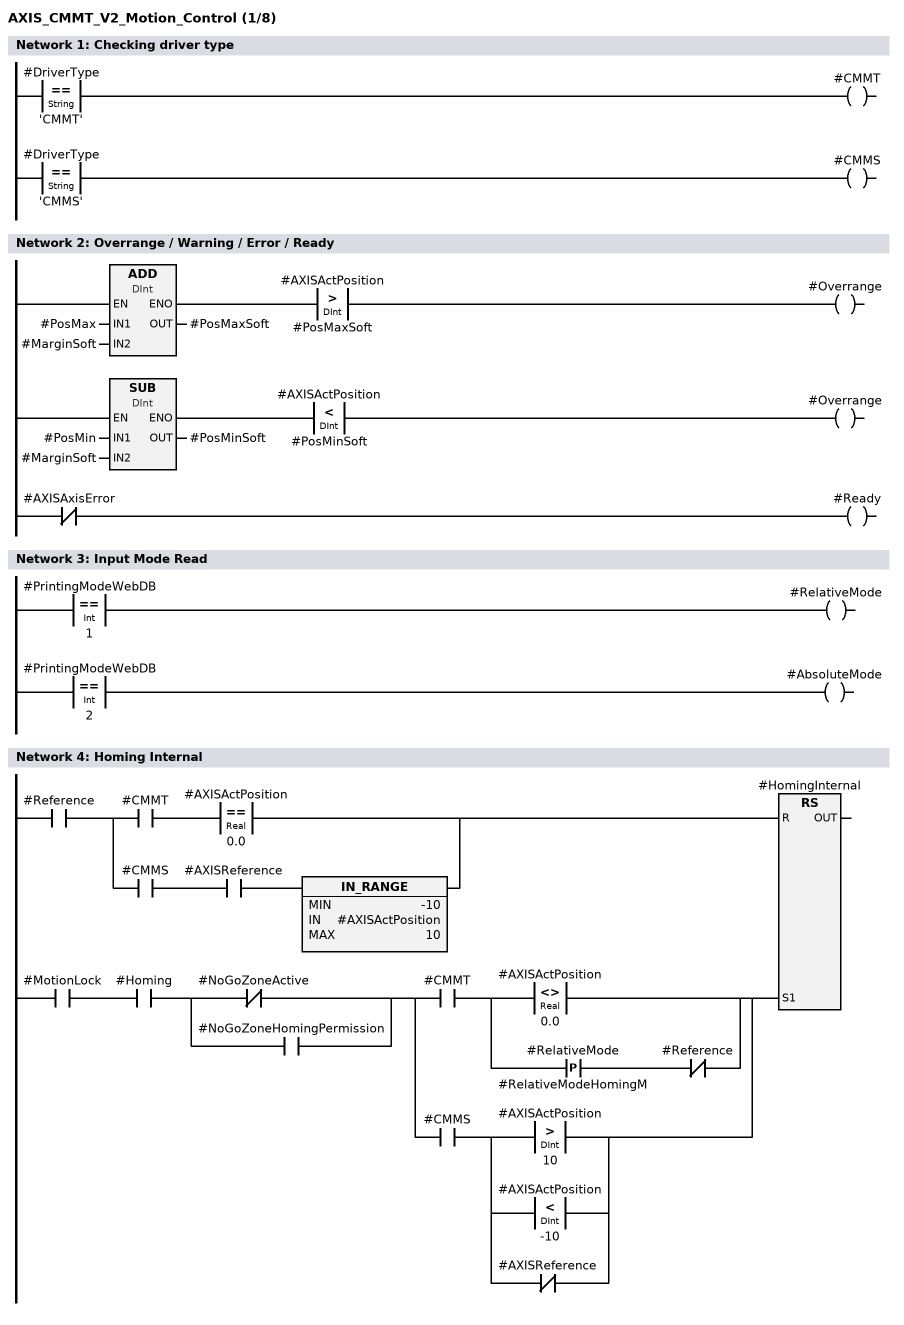
   RUNG wire#powerrail
      { S7_Templates := "SrcType := String" } EQ_Contact(in1 := #DriverType, in2 := 'CMMT')
      Coil( #CMMT )
   END_RUNG
   RUNG wire#powerrail
      { S7_Templates := "SrcType := String" } EQ_Contact(in1 := #DriverType, in2 := 'CMMS')
      Coil( #CMMS )
   END_RUNG
   // the same network as SCL:
   #CMMT := #DriverType = 'CMMT';
   #CMMS := #DriverType = 'CMMS';
END_REGION

REGION Network 2: Overrange / Warning / Error / Ready
   RUNG wire#powerrail
      { S7_Templates := "SrcType := DInt" } Add(in1 := #PosMax, in2 := #MarginSoft, out => #PosMaxSoft)
      { S7_Templates := "SrcType := DInt" } GT_Contact(in1 := #AXISActPosition, in2 := #PosMaxSoft)
      Coil( #Overrange )
   END_RUNG
   RUNG wire#powerrail
      { S7_Templates := "SrcType := DInt" } Sub(in1 := #PosMin, in2 := #MarginSoft, out => #PosMinSoft)
      { S7_Templates := "SrcType := DInt" } LT_Contact(in1 := #AXISActPosition, in2 := #PosMinSoft)
      Coil( #Overrange )
   END_RUNG
   RUNG wire#powerrail
      I_Contact( #AXISAxisError )
      Coil( #Ready )
   END_RUNG
   // the same network as SCL:
   #PosMaxSoft := #PosMax + #MarginSoft;
   #Overrange := #AXISActPosition > #PosMaxSoft;
   #PosMinSoft := #PosMin - #MarginSoft;
   #Overrange := #AXISActPosition < #PosMinSoft;
   #Ready := NOT #AXISAxisError;
END_REGION

REGION Network 3: Input Mode Read
   RUNG wire#powerrail
      { S7_Templates := "SrcType := Int" } EQ_Contact(in1 := #PrintingModeWebDB, in2 := 1)
      Coil( #RelativeMode )
   END_RUNG
   RUNG wire#powerrail
      { S7_Templates := "SrcType := Int" } EQ_Contact(in1 := #PrintingModeWebDB, in2 := 2)
      Coil( #AbsoluteMode )
   END_RUNG
   // the same network as SCL:
   #RelativeMode := #PrintingModeWebDB = 1;
   #AbsoluteMode := #PrintingModeWebDB = 2;
END_REGION

REGION Network 4: Homing Internal
   RUNG wire#powerrail
      Contact( #Reference )
      wire#w1
      Contact( #CMMT )
      { S7_Templates := "SrcType := Real" } EQ_Contact(in1 := #AXISActPosition, in2 := 0.0)
      wire#w2
      S_RS(operand := #HomingInternal, s1 := wire#w7)
   END_RUNG
   RUNG wire#w1
      Contact( #CMMS )
      Contact( #AXISReference )
      { S7_Templates := "SrcType := DInt" } InRange(min := -10, in := #AXISActPosition, max := 10)
   END_RUNG wire#w2
   RUNG wire#powerrail
      Contact( #MotionLock )
      Contact( #Homing )
      wire#w3
      I_Contact( #NoGoZoneActive )
      wire#w4
      Contact( #CMMT )
      wire#w5
      { S7_Templates := "SrcType := Real" } NE_Contact(in1 := #AXISActPosition, in2 := 0.0)
   END_RUNG wire#w7
   RUNG wire#w3
      Contact( #NoGoZoneHomingPermission )
   END_RUNG wire#w4
   RUNG wire#w5
      P_Contact(operand := #RelativeMode, bit := #RelativeModeHomingM)
      I_Contact( #Reference )
   END_RUNG wire#w7
   RUNG wire#w4
      Contact( #CMMS )
      wire#w6
      { S7_Templates := "SrcType := DInt" } GT_Contact(in1 := #AXISActPosition, in2 := 10)
   END_RUNG wire#w7
   RUNG wire#w6
      { S7_Templates := "SrcType := DInt" } LT_Contact(in1 := #AXISActPosition, in2 := -10)
   END_RUNG wire#w7
   RUNG wire#w6
      I_Contact( #AXISReference )
   END_RUNG wire#w7
   // the same network as SCL:
   #_w1 := #MotionLock AND #Homing AND (NOT #NoGoZoneActive OR #NoGoZoneHomingPermission) AND #CMMT AND #RelativeMode AND NOT #RelativeModeHomingM;   // rising edge of #RelativeMode
   #RelativeModeHomingM := #RelativeMode;
   IF #Reference AND ((#CMMT AND (#AXISActPosition = 0.0)) OR (#CMMS AND #AXISReference AND (-10 <= #AXISActPosition) AND (#AXISActPosition <= 10))) THEN
       #HomingInternal := FALSE;   // RS flip-flop
   END_IF;
   IF (#MotionLock AND #Homing AND (NOT #NoGoZoneActive OR #NoGoZoneHomingPermission) AND #CMMT AND (#AXISActPosition <> 0.0)) OR (#_w1 AND NOT #Reference) OR (#MotionLock AND #Homing AND (NOT #NoGoZoneActive OR #NoGoZoneHomingPermission) AND #CMMS AND ((#AXISActPosition > 10) OR (#AXISActPosition < (-10)) OR NOT #AXISReference)) THEN
       #HomingInternal := TRUE;
   END_IF;
END_REGION

REGION Network 5: Status Behavior
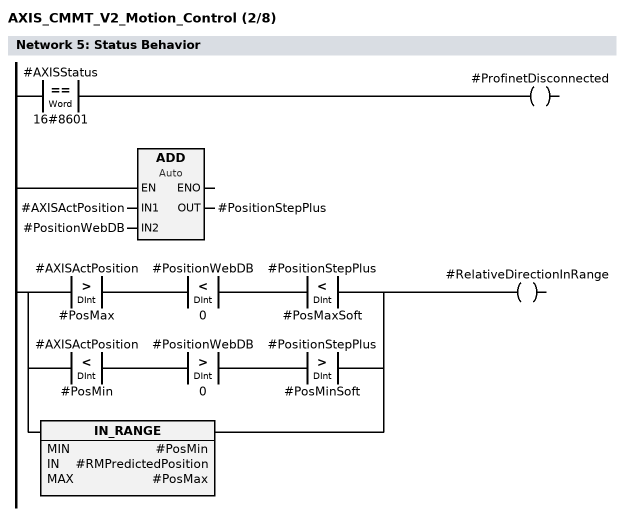
   RUNG wire#powerrail
      { S7_Templates := "SrcType := Word" } EQ_Contact(in1 := #AXISStatus, in2 := 16#8601)
      Coil( #ProfinetDisconnected )
   END_RUNG
   RUNG wire#powerrail
      Add(in1 := #AXISActPosition, in2 := #PositionWebDB, out => #PositionStepPlus)
   END_RUNG
   RUNG wire#powerrail
      { S7_Templates := "SrcType := DInt" } GT_Contact(in1 := #AXISActPosition, in2 := #PosMax)
      { S7_Templates := "SrcType := DInt" } LT_Contact(in1 := #PositionWebDB, in2 := 0)
      { S7_Templates := "SrcType := DInt" } LT_Contact(in1 := #PositionStepPlus, in2 := #PosMaxSoft)
      wire#w1
      Coil( #RelativeDirectionInRange )
   END_RUNG
   RUNG wire#powerrail
      { S7_Templates := "SrcType := DInt" } LT_Contact(in1 := #AXISActPosition, in2 := #PosMin)
      { S7_Templates := "SrcType := DInt" } GT_Contact(in1 := #PositionWebDB, in2 := 0)
      { S7_Templates := "SrcType := DInt" } GT_Contact(in1 := #PositionStepPlus, in2 := #PosMinSoft)
   END_RUNG wire#w1
   RUNG wire#powerrail
      { S7_Templates := "SrcType := DInt" } InRange(min := #PosMin, in := #RMPredictedPosition, max := #PosMax)
   END_RUNG wire#w1
   // the same network as SCL:
   #ProfinetDisconnected := #AXISStatus = 16#8601;
   #PositionStepPlus := #AXISActPosition + #PositionWebDB;
   #RelativeDirectionInRange := ((#AXISActPosition > #PosMax) AND (#PositionWebDB < 0) AND (#PositionStepPlus < #PosMaxSoft)) OR ((#AXISActPosition < #PosMin) AND (#PositionWebDB > 0) AND (#PositionStepPlus > #PosMinSoft)) OR ((#PosMin <= #RMPredictedPosition) AND (#RMPredictedPosition <= #PosMax));
END_REGION

REGION Network 6: Task Internal
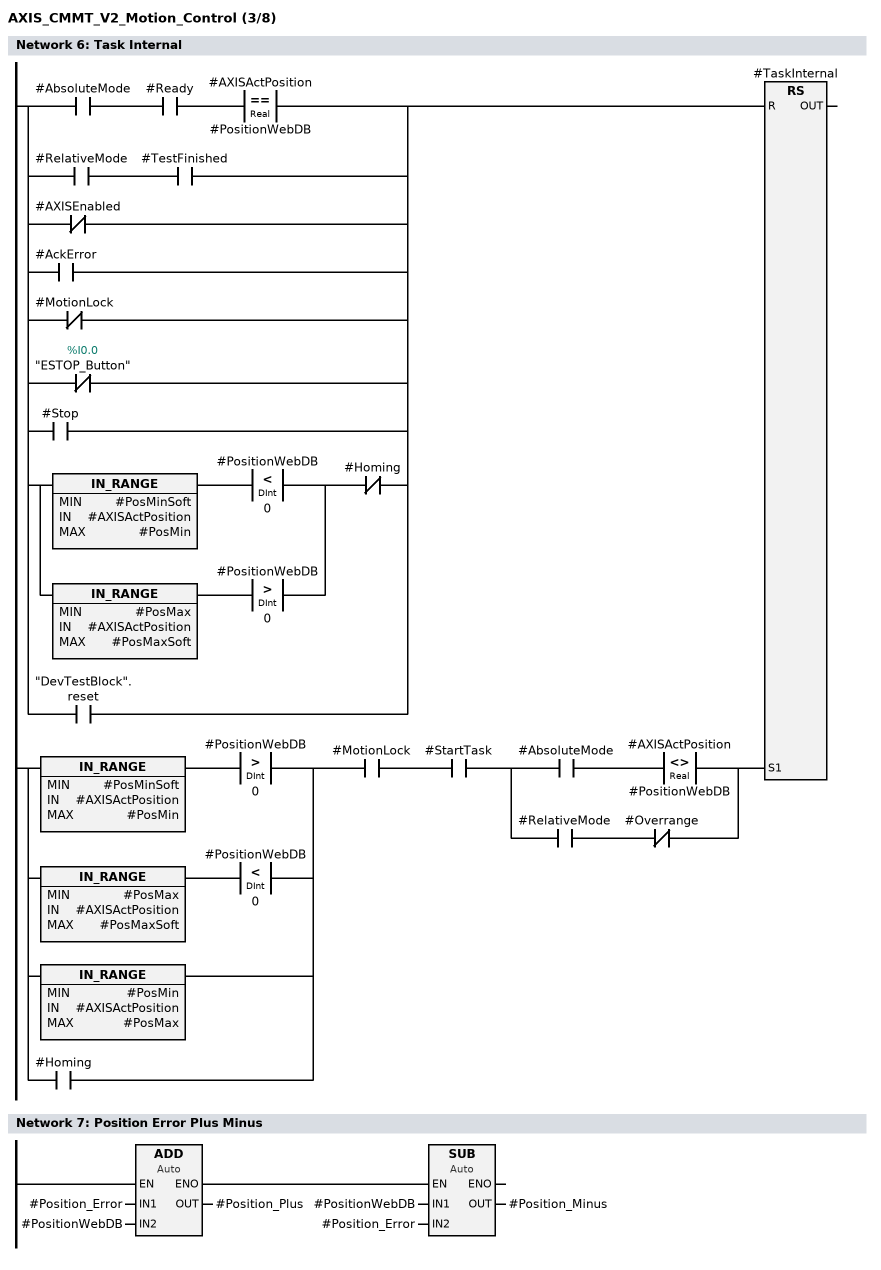
   RUNG wire#powerrail
      Contact( #AbsoluteMode )
      Contact( #Ready )
      { S7_Templates := "SrcType := Real" } EQ_Contact(in1 := #AXISActPosition, in2 := #PositionWebDB)
      wire#w1
      S_RS(operand := #TaskInternal, s1 := wire#w5)
   END_RUNG
   RUNG wire#powerrail
      Contact( #RelativeMode )
      Contact( #TestFinished )
   END_RUNG wire#w1
   RUNG wire#powerrail
      I_Contact( #AXISEnabled )
   END_RUNG wire#w1
   RUNG wire#powerrail
      Contact( #AckError )
   END_RUNG wire#w1
   RUNG wire#powerrail
      I_Contact( #MotionLock )
   END_RUNG wire#w1
   RUNG wire#powerrail
      I_Contact( "ESTOP_Button" )
   END_RUNG wire#w1
   RUNG wire#powerrail
      Contact( #Stop )
   END_RUNG wire#w1
   RUNG wire#powerrail
      { S7_Templates := "SrcType := DInt" } InRange(min := #PosMinSoft, in := #AXISActPosition, max := #PosMin)
      { S7_Templates := "SrcType := DInt" } LT_Contact(in1 := #PositionWebDB, in2 := 0)
      wire#w2
      I_Contact( #Homing )
   END_RUNG wire#w1
   RUNG wire#powerrail
      { S7_Templates := "SrcType := DInt" } InRange(min := #PosMax, in := #AXISActPosition, max := #PosMaxSoft)
      { S7_Templates := "SrcType := DInt" } GT_Contact(in1 := #PositionWebDB, in2 := 0)
   END_RUNG wire#w2
   RUNG wire#powerrail
      Contact( "DevTestBlock".reset )
   END_RUNG wire#w1
   RUNG wire#powerrail
      { S7_Templates := "SrcType := DInt" } InRange(min := #PosMinSoft, in := #AXISActPosition, max := #PosMin)
      { S7_Templates := "SrcType := DInt" } GT_Contact(in1 := #PositionWebDB, in2 := 0)
      wire#w3
      Contact( #MotionLock )
      Contact( #StartTask )
      wire#w4
      Contact( #AbsoluteMode )
      { S7_Templates := "SrcType := Real" } NE_Contact(in1 := #AXISActPosition, in2 := #PositionWebDB)
   END_RUNG wire#w5
   RUNG wire#powerrail
      { S7_Templates := "SrcType := DInt" } InRange(min := #PosMax, in := #AXISActPosition, max := #PosMaxSoft)
      { S7_Templates := "SrcType := DInt" } LT_Contact(in1 := #PositionWebDB, in2 := 0)
   END_RUNG wire#w3
   RUNG wire#powerrail
      { S7_Templates := "SrcType := DInt" } InRange(min := #PosMin, in := #AXISActPosition, max := #PosMax)
   END_RUNG wire#w3
   RUNG wire#powerrail
      Contact( #Homing )
   END_RUNG wire#w3
   RUNG wire#w4
      Contact( #RelativeMode )
      I_Contact( #Overrange )
   END_RUNG wire#w5
   // the same network as SCL:
   IF (#AbsoluteMode AND #Ready AND (#AXISActPosition = #PositionWebDB)) OR (#RelativeMode AND #TestFinished) OR NOT #AXISEnabled OR #AckError OR NOT #MotionLock OR NOT "ESTOP_Button" OR #Stop OR ((((#PosMinSoft <= #AXISActPosition) AND (#AXISActPosition <= #PosMin) AND (#PositionWebDB < 0)) OR ((#PosMax <= #AXISActPosition) AND (#AXISActPosition <= #PosMaxSoft) AND (#PositionWebDB > 0))) AND NOT #Homing) OR "DevTestBlock".reset THEN
       #TaskInternal := FALSE;   // RS flip-flop
   END_IF;
   IF (((#PosMinSoft <= #AXISActPosition) AND (#AXISActPosition <= #PosMin) AND (#PositionWebDB > 0)) OR ((#PosMax <= #AXISActPosition) AND (#AXISActPosition <= #PosMaxSoft) AND (#PositionWebDB < 0)) OR ((#PosMin <= #AXISActPosition) AND (#AXISActPosition <= #PosMax)) OR #Homing) AND #MotionLock AND #StartTask AND ((#AbsoluteMode AND (#AXISActPosition <> #PositionWebDB)) OR (#RelativeMode AND NOT #Overrange)) THEN
       #TaskInternal := TRUE;
   END_IF;
END_REGION

REGION Network 7: Position Error Plus Minus
   RUNG wire#powerrail
      Add(in1 := #Position_Error, in2 := #PositionWebDB, out => #Position_Plus)
      Sub(in1 := #PositionWebDB, in2 := #Position_Error, out => #Position_Minus)
   END_RUNG
   // the same network as SCL:
   #Position_Plus := #Position_Error + #PositionWebDB;
   #Position_Minus := #PositionWebDB - #Position_Error;
END_REGION

REGION Network 8: Execute Internal
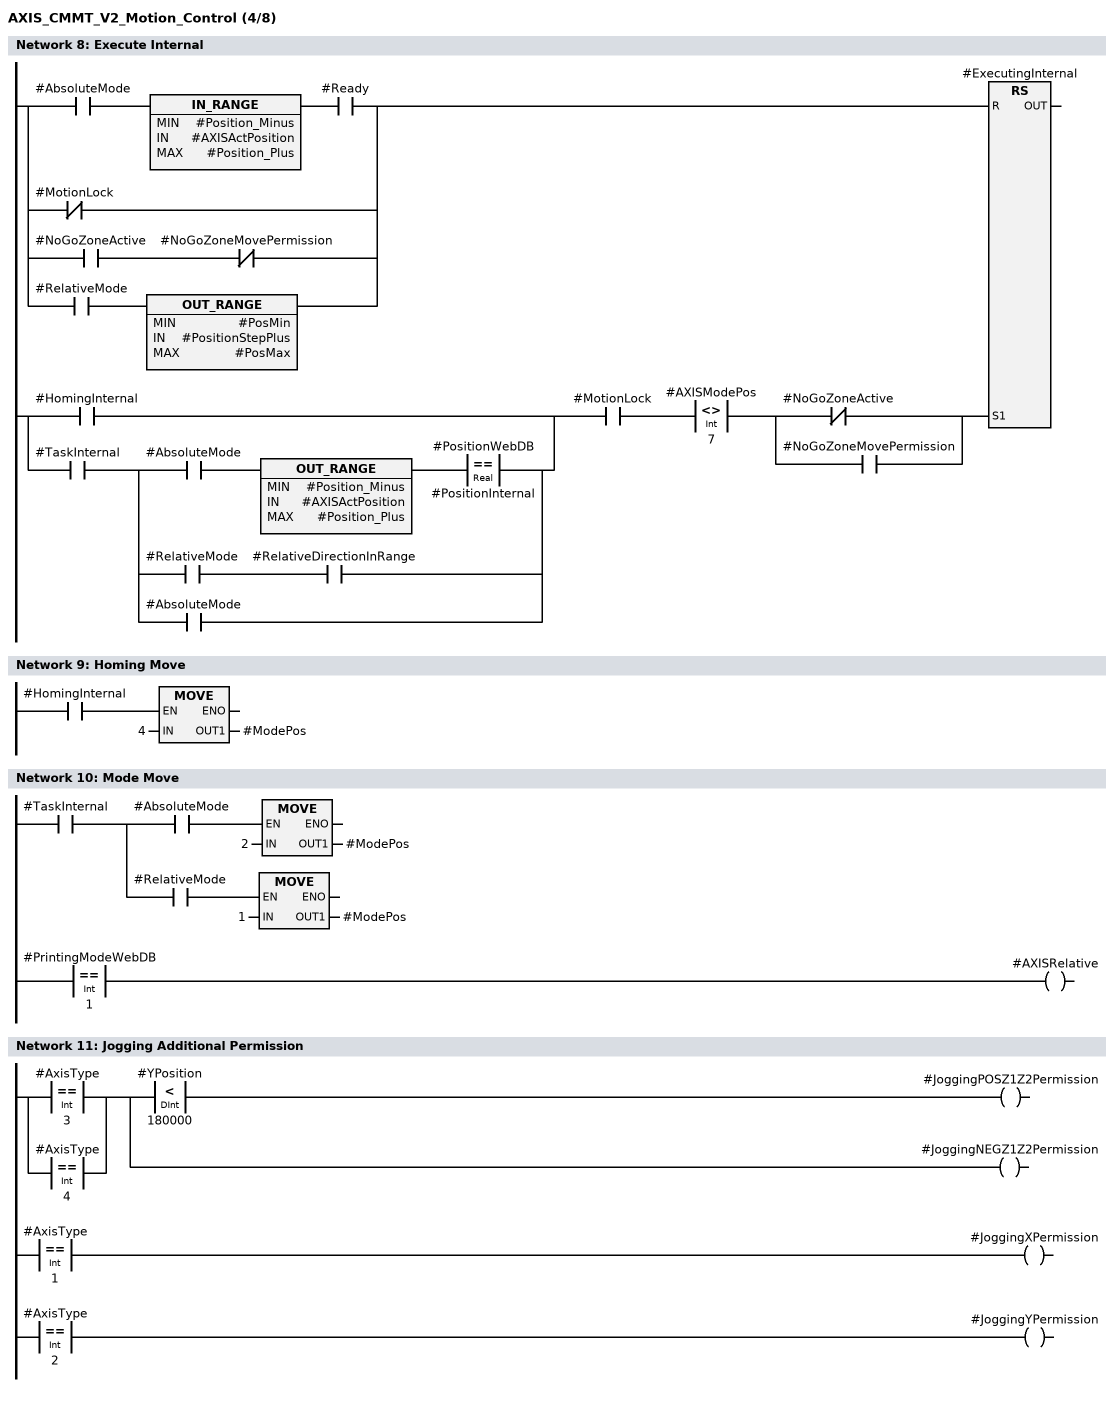
   IF (#AbsoluteMode AND (#Position_Minus <= #AXISActPosition) AND (#AXISActPosition <= #Position_Plus) AND #Ready) OR NOT #MotionLock OR (#NoGoZoneActive AND NOT #NoGoZoneMovePermission) OR (#RelativeMode AND ((#PositionStepPlus < #PosMin) OR (#PositionStepPlus > #PosMax))) THEN
       #ExecutingInternal := FALSE;   // RS flip-flop
   END_IF;
   IF (#HomingInternal OR (#TaskInternal AND ((#AbsoluteMode AND ((#AXISActPosition < #Position_Minus) OR (#AXISActPosition > #Position_Plus)) AND (#PositionWebDB = #PositionInternal)) OR (#RelativeMode AND #RelativeDirectionInRange) OR #AbsoluteMode))) AND #MotionLock AND (#AXISModePos <> 7) AND (NOT #NoGoZoneActive OR #NoGoZoneMovePermission) THEN
       #ExecutingInternal := TRUE;
   END_IF;
END_REGION

REGION Network 9: Homing Move
   RUNG wire#powerrail
      Contact( #HomingInternal )
      Move(in := 4, out1 => #ModePos)
   END_RUNG
   // the same network as SCL:
   IF #HomingInternal THEN #ModePos := 4; END_IF;
END_REGION

REGION Network 10: Mode Move
   RUNG wire#powerrail
      Contact( #TaskInternal )
      wire#w1
      Contact( #AbsoluteMode )
      Move(in := 2, out1 => #ModePos)
   END_RUNG
   RUNG wire#w1
      Contact( #RelativeMode )
      Move(in := 1, out1 => #ModePos)
   END_RUNG
   RUNG wire#powerrail
      { S7_Templates := "SrcType := Int" } EQ_Contact(in1 := #PrintingModeWebDB, in2 := 1)
      Coil( #AXISRelative )
   END_RUNG
   // the same network as SCL:
   IF #TaskInternal AND #AbsoluteMode THEN #ModePos := 2; END_IF;
   IF #TaskInternal AND #RelativeMode THEN #ModePos := 1; END_IF;
   #AXISRelative := #PrintingModeWebDB = 1;
END_REGION

REGION Network 11: Jogging Additional Permission
   RUNG wire#powerrail
      { S7_Templates := "SrcType := Int" } EQ_Contact(in1 := #AxisType, in2 := 3)
      wire#w1
      { S7_Templates := "SrcType := DInt" } LT_Contact(in1 := #YPosition, in2 := 180000)
      Coil( #JoggingPOSZ1Z2Permission )
   END_RUNG
   RUNG wire#powerrail
      { S7_Templates := "SrcType := Int" } EQ_Contact(in1 := #AxisType, in2 := 4)
   END_RUNG wire#w1
   RUNG wire#w1
      Coil( #JoggingNEGZ1Z2Permission )
   END_RUNG
   RUNG wire#powerrail
      { S7_Templates := "SrcType := Int" } EQ_Contact(in1 := #AxisType, in2 := 1)
      Coil( #JoggingXPermission )
   END_RUNG
   RUNG wire#powerrail
      { S7_Templates := "SrcType := Int" } EQ_Contact(in1 := #AxisType, in2 := 2)
      Coil( #JoggingYPermission )
   END_RUNG
   // the same network as SCL:
   #_w1 := (#AxisType = 3) OR (#AxisType = 4);
   #JoggingPOSZ1Z2Permission := #_w1 AND (#YPosition < 180000);
   #JoggingNEGZ1Z2Permission := #_w1;
   #JoggingXPermission := #AxisType = 1;
   #JoggingYPermission := #AxisType = 2;
END_REGION

REGION Network 12: Jogging Limit Change
   // Changed jogging limits to prevent overshooting
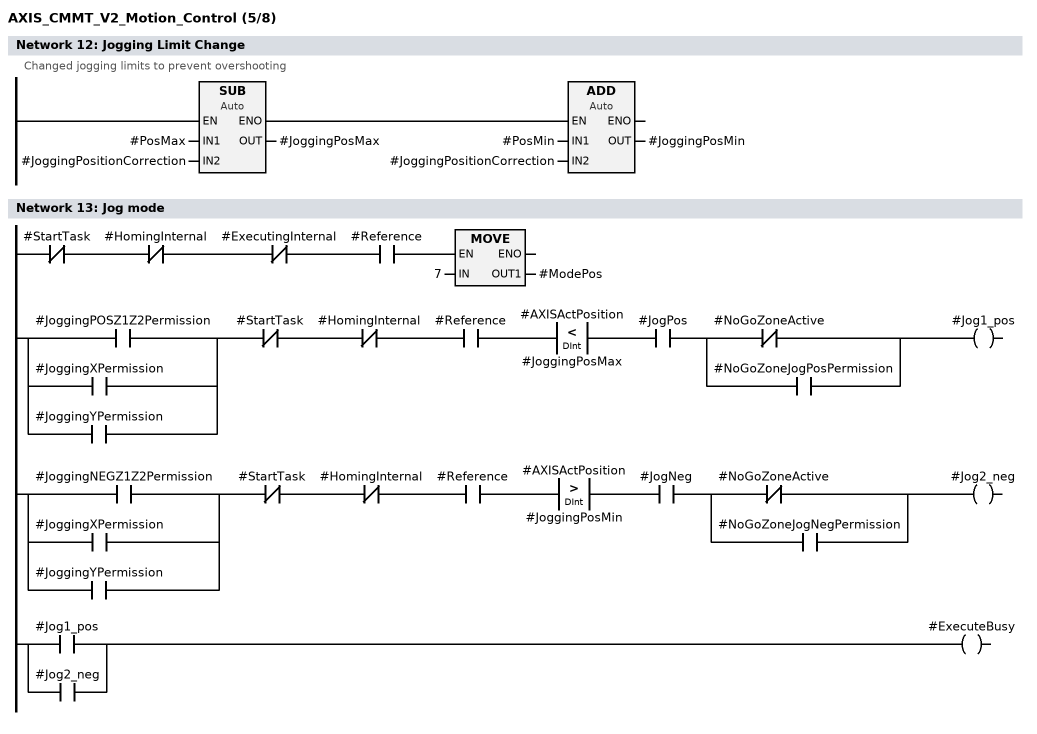
   RUNG wire#powerrail
      Sub(in1 := #PosMax, in2 := #JoggingPositionCorrection, out => #JoggingPosMax)
      Add(in1 := #PosMin, in2 := #JoggingPositionCorrection, out => #JoggingPosMin)
   END_RUNG
   // the same network as SCL:
   #JoggingPosMax := #PosMax - #JoggingPositionCorrection;
   #JoggingPosMin := #PosMin + #JoggingPositionCorrection;
END_REGION

REGION Network 13: Jog mode
   RUNG wire#powerrail
      I_Contact( #StartTask )
      I_Contact( #HomingInternal )
      I_Contact( #ExecutingInternal )
      Contact( #Reference )
      Move(in := 7, out1 => #ModePos)
   END_RUNG
   RUNG wire#powerrail
      Contact( #JoggingPOSZ1Z2Permission )
      wire#w1
      I_Contact( #StartTask )
      I_Contact( #HomingInternal )
      Contact( #Reference )
      { S7_Templates := "SrcType := DInt" } LT_Contact(in1 := #AXISActPosition, in2 := #JoggingPosMax)
      Contact( #JogPos )
      wire#w2
      I_Contact( #NoGoZoneActive )
      wire#w3
      Coil( #Jog1_pos )
   END_RUNG
   RUNG wire#powerrail
      Contact( #JoggingXPermission )
   END_RUNG wire#w1
   RUNG wire#powerrail
      Contact( #JoggingYPermission )
   END_RUNG wire#w1
   RUNG wire#w2
      Contact( #NoGoZoneJogPosPermission )
   END_RUNG wire#w3
   RUNG wire#powerrail
      Contact( #JoggingNEGZ1Z2Permission )
      wire#w4
      I_Contact( #StartTask )
      I_Contact( #HomingInternal )
      Contact( #Reference )
      { S7_Templates := "SrcType := DInt" } GT_Contact(in1 := #AXISActPosition, in2 := #JoggingPosMin)
      Contact( #JogNeg )
      wire#w5
      I_Contact( #NoGoZoneActive )
      wire#w6
      Coil( #Jog2_neg )
   END_RUNG
   RUNG wire#powerrail
      Contact( #JoggingXPermission )
   END_RUNG wire#w4
   RUNG wire#powerrail
      Contact( #JoggingYPermission )
   END_RUNG wire#w4
   RUNG wire#w5
      Contact( #NoGoZoneJogNegPermission )
   END_RUNG wire#w6
   RUNG wire#powerrail
      Contact( #Jog1_pos )
      wire#w7
      Coil( #ExecuteBusy )
   END_RUNG
   RUNG wire#powerrail
      Contact( #Jog2_neg )
   END_RUNG wire#w7
   // the same network as SCL:
   IF NOT #StartTask AND NOT #HomingInternal AND NOT #ExecutingInternal AND #Reference THEN
       #ModePos := 7;
   END_IF;
   #Jog1_pos := (#JoggingPOSZ1Z2Permission OR #JoggingXPermission OR #JoggingYPermission) AND NOT #StartTask AND NOT #HomingInternal AND #Reference AND (#AXISActPosition < #JoggingPosMax) AND #JogPos AND (NOT #NoGoZoneActive OR #NoGoZoneJogPosPermission);
   #Jog2_neg := (#JoggingNEGZ1Z2Permission OR #JoggingXPermission OR #JoggingYPermission) AND NOT #StartTask AND NOT #HomingInternal AND #Reference AND (#AXISActPosition > #JoggingPosMin) AND #JogNeg AND (NOT #NoGoZoneActive OR #NoGoZoneJogNegPermission);
   #ExecuteBusy := #Jog1_pos OR #Jog2_neg;
END_REGION

REGION Network 14: Motion Block Control
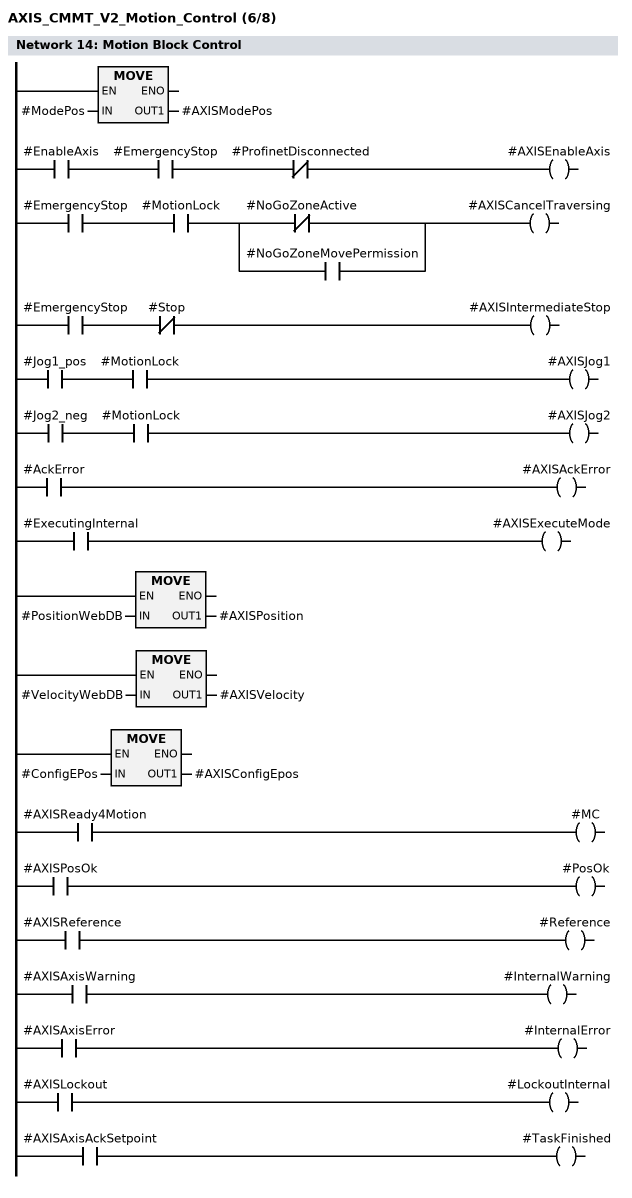
   RUNG wire#powerrail
      Move(in := #ModePos, out1 => #AXISModePos)
   END_RUNG
   RUNG wire#powerrail
      Contact( #EnableAxis )
      Contact( #EmergencyStop )
      I_Contact( #ProfinetDisconnected )
      Coil( #AXISEnableAxis )
   END_RUNG
   RUNG wire#powerrail
      Contact( #EmergencyStop )
      Contact( #MotionLock )
      wire#w1
      I_Contact( #NoGoZoneActive )
      wire#w2
      Coil( #AXISCancelTraversing )
   END_RUNG
   RUNG wire#w1
      Contact( #NoGoZoneMovePermission )
   END_RUNG wire#w2
   RUNG wire#powerrail
      Contact( #EmergencyStop )
      I_Contact( #Stop )
      Coil( #AXISIntermediateStop )
   END_RUNG
   RUNG wire#powerrail
      Contact( #Jog1_pos )
      Contact( #MotionLock )
      Coil( #AXISJog1 )
   END_RUNG
   RUNG wire#powerrail
      Contact( #Jog2_neg )
      Contact( #MotionLock )
      Coil( #AXISJog2 )
   END_RUNG
   RUNG wire#powerrail
      Contact( #AckError )
      Coil( #AXISAckError )
   END_RUNG
   RUNG wire#powerrail
      Contact( #ExecutingInternal )
      Coil( #AXISExecuteMode )
   END_RUNG
   RUNG wire#powerrail
      Move(in := #PositionWebDB, out1 => #AXISPosition)
   END_RUNG
   RUNG wire#powerrail
      Move(in := #VelocityWebDB, out1 => #AXISVelocity)
   END_RUNG
   RUNG wire#powerrail
      Move(in := #ConfigEPos, out1 => #AXISConfigEpos)
   END_RUNG
   RUNG wire#powerrail
      Contact( #AXISReady4Motion )
      Coil( #MC )
   END_RUNG
   RUNG wire#powerrail
      Contact( #AXISPosOk )
      Coil( #PosOk )
   END_RUNG
   RUNG wire#powerrail
      Contact( #AXISReference )
      Coil( #Reference )
   END_RUNG
   RUNG wire#powerrail
      Contact( #AXISAxisWarning )
      Coil( #InternalWarning )
   END_RUNG
   RUNG wire#powerrail
      Contact( #AXISAxisError )
      Coil( #InternalError )
   END_RUNG
   RUNG wire#powerrail
      Contact( #AXISLockout )
      Coil( #LockoutInternal )
   END_RUNG
   RUNG wire#powerrail
      Contact( #AXISAxisAckSetpoint )
      Coil( #TaskFinished )
   END_RUNG
   // the same network as SCL:
   #AXISModePos := #ModePos;
   #AXISEnableAxis := #EnableAxis AND #EmergencyStop AND NOT #ProfinetDisconnected;
   #AXISCancelTraversing := #EmergencyStop AND #MotionLock AND (NOT #NoGoZoneActive OR #NoGoZoneMovePermission);
   #AXISIntermediateStop := #EmergencyStop AND NOT #Stop;
   #AXISJog1 := #Jog1_pos AND #MotionLock;
   #AXISJog2 := #Jog2_neg AND #MotionLock;
   #AXISAckError := #AckError;
   #AXISExecuteMode := #ExecutingInternal;
   #AXISPosition := #PositionWebDB;
   #AXISVelocity := #VelocityWebDB;
   #AXISConfigEpos := #ConfigEPos;
   #MC := #AXISReady4Motion;
   #PosOk := #AXISPosOk;
   #Reference := #AXISReference;
   #InternalWarning := #AXISAxisWarning;
   #InternalError := #AXISAxisError;
   #LockoutInternal := #AXISLockout;
   #TaskFinished := #AXISAxisAckSetpoint;
END_REGION

REGION Network 15: Mem
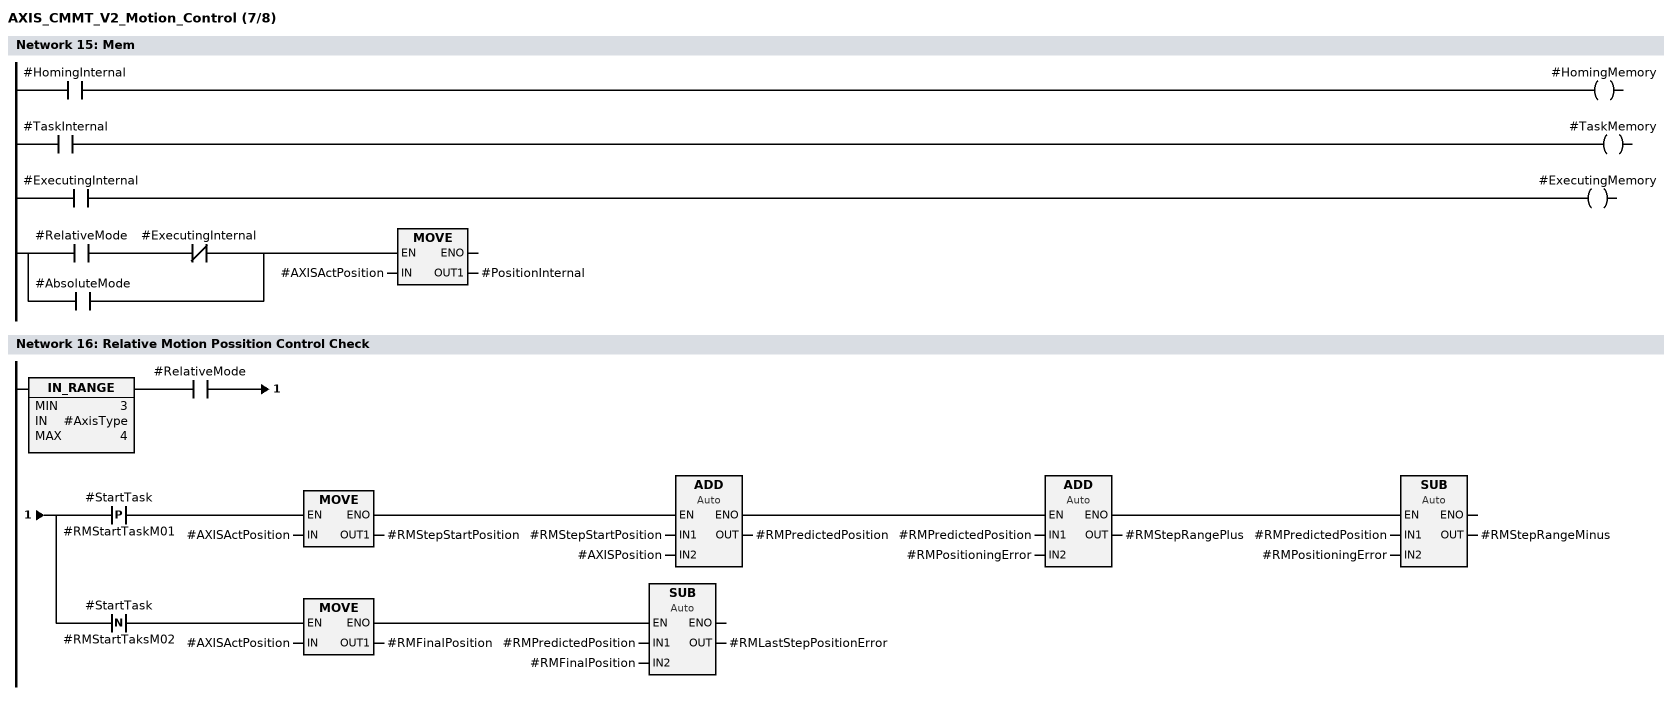
   RUNG wire#powerrail
      Contact( #HomingInternal )
      Coil( #HomingMemory )
   END_RUNG
   RUNG wire#powerrail
      Contact( #TaskInternal )
      Coil( #TaskMemory )
   END_RUNG
   RUNG wire#powerrail
      Contact( #ExecutingInternal )
      Coil( #ExecutingMemory )
   END_RUNG
   RUNG wire#powerrail
      Contact( #RelativeMode )
      I_Contact( #ExecutingInternal )
      wire#w1
      Move(in := #AXISActPosition, out1 => #PositionInternal)
   END_RUNG
   RUNG wire#powerrail
      Contact( #AbsoluteMode )
   END_RUNG wire#w1
   // the same network as SCL:
   #HomingMemory := #HomingInternal;
   #TaskMemory := #TaskInternal;
   #ExecutingMemory := #ExecutingInternal;
   IF (#RelativeMode AND NOT #ExecutingInternal) OR #AbsoluteMode THEN
       #PositionInternal := #AXISActPosition;
   END_IF;
END_REGION

REGION Network 16: Relative Motion Possition Control Check
   RUNG wire#powerrail
      { S7_Templates := "SrcType := Int" } InRange(min := 3, in := #AxisType, max := 4)
      Contact( #RelativeMode )
      wire#w1
      P_Contact(operand := #StartTask, bit := #RMStartTaskM01)
      Move(in := #AXISActPosition, out1 => #RMStepStartPosition)
      Add(in1 := #RMStepStartPosition, in2 := #AXISPosition, out => #RMPredictedPosition)
      Add(in1 := #RMPredictedPosition, in2 := #RMPositioningError, out => #RMStepRangePlus)
      Sub(in1 := #RMPredictedPosition, in2 := #RMPositioningError, out => #RMStepRangeMinus)
   END_RUNG
   RUNG wire#w1
      N_Contact(operand := #StartTask, bit := #RMStartTaksM02)
      Move(in := #AXISActPosition, out1 => #RMFinalPosition)
      Sub(in1 := #RMPredictedPosition, in2 := #RMFinalPosition, out => #RMLastStepPositionError)
   END_RUNG
   // the same network as SCL:
   #_w1 := (3 <= #AxisType) AND (#AxisType <= 4) AND #RelativeMode;
   #_w2 := #_w1 AND #StartTask AND NOT #RMStartTaskM01;   // rising edge of #StartTask
   #RMStartTaskM01 := #StartTask;
   IF #_w2 THEN
       #RMStepStartPosition := #AXISActPosition;
       #RMPredictedPosition := #RMStepStartPosition + #AXISPosition;
       #RMStepRangePlus := #RMPredictedPosition + #RMPositioningError;
       #RMStepRangeMinus := #RMPredictedPosition - #RMPositioningError;
   END_IF;
   #_w3 := #_w1 AND NOT #StartTask AND #RMStartTaksM02;   // falling edge of #StartTask
   #RMStartTaksM02 := #StartTask;
   IF #_w3 THEN
       #RMFinalPosition := #AXISActPosition;
       #RMLastStepPositionError := #RMPredictedPosition - #RMFinalPosition;
   END_IF;
END_REGION

REGION Network 17: Status Move
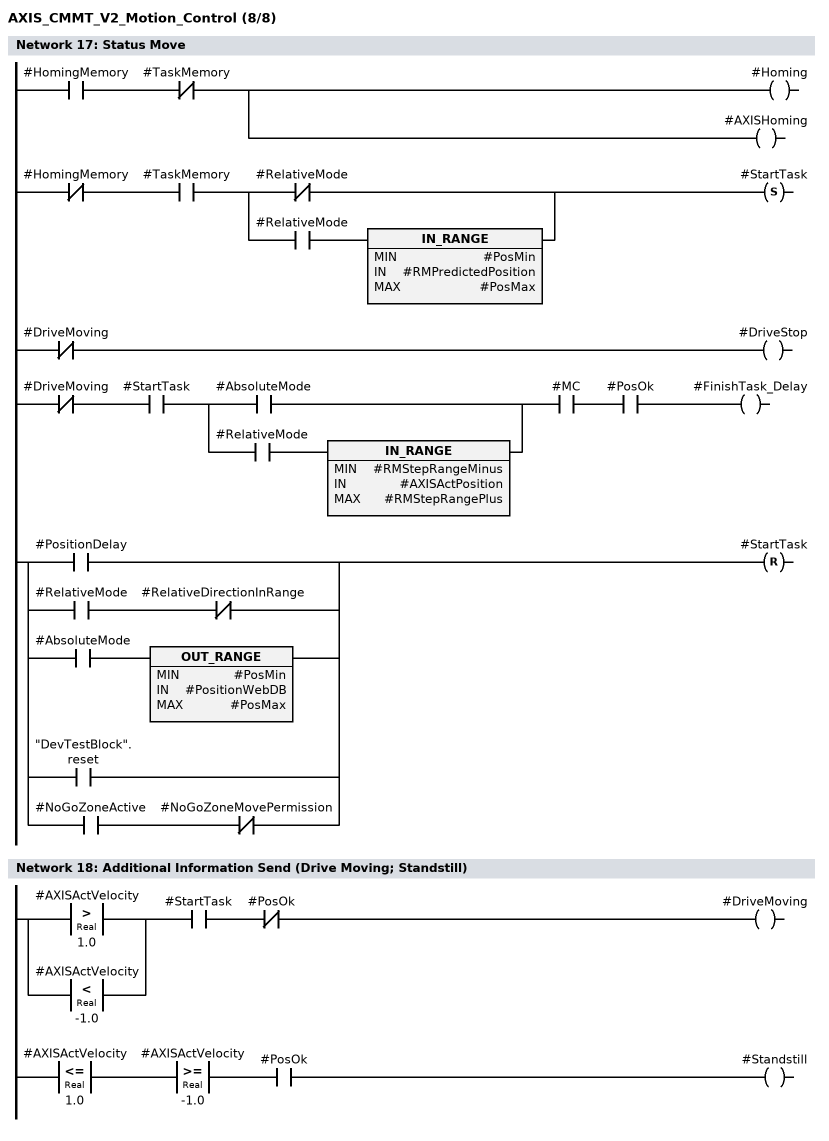
   #Homing := #HomingMemory AND NOT #TaskMemory;
   #AXISHoming := #Homing;
   IF NOT #HomingMemory AND #TaskMemory AND (NOT #RelativeMode OR (#RelativeMode AND (#PosMin <= #RMPredictedPosition) AND (#RMPredictedPosition <= #PosMax))) THEN
       #StartTask := TRUE;
   END_IF;
   #DriveStop := NOT #DriveMoving;
   #FinishTask_Delay := NOT #DriveMoving AND #StartTask AND (#AbsoluteMode OR (#RelativeMode AND (#RMStepRangeMinus <= #AXISActPosition) AND (#AXISActPosition <= #RMStepRangePlus))) AND #MC AND #PosOk;
   IF #PositionDelay OR (#RelativeMode AND NOT #RelativeDirectionInRange) OR (#AbsoluteMode AND ((#PositionWebDB < #PosMin) OR (#PositionWebDB > #PosMax))) OR "DevTestBlock".reset OR (#NoGoZoneActive AND NOT #NoGoZoneMovePermission) THEN
       #StartTask := FALSE;
   END_IF;
END_REGION

REGION Network 18: Additional Information Send (Drive Moving; Standstill)
   RUNG wire#powerrail
      { S7_Templates := "SrcType := Real" } GT_Contact(in1 := #AXISActVelocity, in2 := 1.0)
      wire#w1
      Contact( #StartTask )
      I_Contact( #PosOk )
      Coil( #DriveMoving )
   END_RUNG
   RUNG wire#powerrail
      { S7_Templates := "SrcType := Real" } LT_Contact(in1 := #AXISActVelocity, in2 := -1.0)
   END_RUNG wire#w1
   RUNG wire#powerrail
      { S7_Templates := "SrcType := Real" } LE_Contact(in1 := #AXISActVelocity, in2 := 1.0)
      { S7_Templates := "SrcType := Real" } GE_Contact(in1 := #AXISActVelocity, in2 := -1.0)
      Contact( #PosOk )
      Coil( #Standstill )
   END_RUNG
   // the same network as SCL:
   #DriveMoving := ((#AXISActVelocity > 1.0) OR (#AXISActVelocity < (-1.0))) AND #StartTask AND NOT #PosOk;
   #Standstill := (#AXISActVelocity <= 1.0) AND (#AXISActVelocity >= (-1.0)) AND #PosOk;
END_REGION
END_FUNCTION_BLOCK

FUNCTION_BLOCK "Festo_PtP_Drives_PN"
{ S7_Optimized_Access := 'TRUE' }
AUTHOR : Festo
FAMILY : 'E-.Drives'
VERSION : 1.5
   VAR_INPUT 
      ModePos : Int := 0;
      EnableAxis : Bool := 0;
      CancelTraversing : Bool := 1;
      IntermediateStop : Bool := 1;
      Positive : Bool := 0;
      Negative : Bool := 0;
      Jog1 : Bool := 0;
      Jog2 : Bool := 0;
      AckError : Bool := 0;
      ExecuteMode : Bool := 0;
      ReleaseBrake : Bool := 0;
      TravelToFixStop : Bool := 0;
      Position : DInt := 0;
      Velocity : DInt := 0;
      OverV : Int := 100;
      OverAcc : Int := 100;
      OverDec : Int := 100;
      ConfigEPos : DWord := 16#0000_000F;
      BaseSpeedValue : Real;
      HardwareId : HW_IO := 0;
   END_VAR

   VAR_OUTPUT 
      AxisEnabled : Bool := 0;
      AxisPosOk : Bool := 0;
      AxisSpFixed : Bool := 0;
      AxisAckSetpoint : Bool := 0;
      ClampTorqueReached : Bool;
      AxisRef : Bool := 0;
      AxisWarn : Bool := 0;
      AxisError : Bool := 0;
      Lockout : Bool := 0;
      ActVelocity : Real := 0.0;
      ActPosition : DInt := 0;
      ActMode : Int := 0;
      EPosZSW1 : Word := 0;
      EPosZSW2 : Word := 0;
      ActWarn : Word := 0;
      ActFault : Word := 0;
      Error : Bool := 0;
      Status : Word := 0;
      DiagID : Word := 0;
   END_VAR

   VAR 
      stat_Ready4Motion : Bool := 0;
      stat_ExecuteIntern : Bool := 0;
      stat_StepHome : UInt;
      stat_RetDPRD : Int;
      stat_RetDPWR : Int;
      stat_CycWrite : Struct
         STW1 : Struct
            jog1 : Bool;
            jog2 : Bool;
            controlByPlc : Bool := TRUE;
            StartHoming : Bool;
            ReleaseBrake : Bool;
            ExternalBlockChange : Bool;
            reserved14 : Bool;
            reserved15 : Bool;
            on : Bool;
            noCoastStop : Bool := TRUE;
            noQuickStop : Bool := TRUE;
            enableOperation : Bool := TRUE;
            cancelTraversing : Bool;
            intermediateStop : Bool;
            activateTraversing : Bool;
            acknowledgeFault : Bool;
         END_STRUCT;
         POS_STW1 : Struct
            MDI_MOD : Bool;
            PosModulo : Bool;
            NegModulo : Bool;
            reserved11 : Bool;
            reserved12 : Bool;
            reserved13 : Bool;
            SetupMode : Bool;
            MDI_Activate : Bool;
            travBlockBit0 : Bool;
            travBlockBit1 : Bool;
            travBlockBit2 : Bool;
            travBlockBit3 : Bool;
            travBlockBit4 : Bool;
            travBlockBit5 : Bool;
            travBlockBit6 : Bool;
            reserved7 : Bool;
         END_STRUCT;
         POS_STW2 : Struct
            FlyingRef : Bool;
            reserved9 : Bool;
            SelectProbe : Bool;
            ProbeEdgeEval : Bool;
            reserved12 : Bool;
            reserved13 : Bool;
            "SW-Limit" : Bool;
            "HW-Limit" : Bool;
            Trackingmode : Bool;
            SetReferencePoint : Bool;
            reserved2 : Bool;
            reserved3 : Bool;
            reserved4 : Bool;
            jog_inc : Bool;
            reserved6 : Bool;
            reserved7 : Bool;
         END_STRUCT;
         STW2 : Struct
            TravelToFixStop : Bool;
            reserved9 : Bool;
            reserved10 : Bool;
            reserved11 : Bool;
            signOfLifeBit0 : Bool;
            signOfLifeBit1 : Bool;
            signOfLifeBit2 : Bool;
            signOfLifeBit3 : Bool;
            reserved0 : Bool;
            reserved1 : Bool;
            reserved2 : Bool;
            reserved3 : Bool;
            reserved4 : Bool;
            reserved5 : Bool;
            reserved6 : Bool;
            reserved7 : Bool;
         END_STRUCT;
         Override : Word;
         MDI_TARPOS : DInt;
         MDI_VELOCITY : DInt;
         MDI_ACC : UInt;
         MDI_DEC : UInt;
         reserved11 : Word;
      END_STRUCT;
      stat_CycRead : Struct
         ZSW1 : Struct
            followingErrorInTolerance : Bool;
            controlRequest : Bool;
            targetPosReached : Bool;
            homePosSet : Bool;
            acknowledgeTraversingBlockActivated : Bool;
            driveStopped : Bool;
            axisAccelerates : Bool;
            axisDecelerates : Bool;
            readyForSwitchOn : Bool;
            ready : Bool;
            operationEnabled : Bool;
            faultPresent : Bool;
            noCoastingActive : Bool;
            noQuickStopActive : Bool;
            switchingOnInhibitedActive : Bool;
            warningActive : Bool;
         END_STRUCT;
         POS_ZSW1 : Word;
         POS_ZSW2 : Word;
         ZSW2 : Struct
            deviceSpecificBit8 : Bool;
            deviceSpecificBit9 : Bool;
            deviceSpecificBit10 : Bool;
            deviceSpecificBit11 : Bool;
            doSignOfLifeBit0 : Bool;
            doSignOfLifeBit1 : Bool;
            doSignOfLifeBit2 : Bool;
            doSignOfLifeBit3 : Bool;
            deviceSpecificBit0 : Bool;
            deviceSpecificBit1 : Bool;
            deviceSpecificBit2 : Bool;
            deviceSpecificBit3 : Bool;
            deviceSpecificBit4 : Bool;
            deviceSpecificBit5 : Bool;
            deviceSpecificBit6 : Bool;
            deviceSpecificBit7 : Bool;
         END_STRUCT;
         MELDW : Word;
         XIST_A : DInt;
         NIST_B : DInt;
         Fault_Code : Word;
         Warn_Code : Word;
         Reserved : Word;
      END_STRUCT;
      stat_ExecAux : Bool;
      stat_ExecR_Trig : Bool;
      stat_Jog1PAux : Bool;
      stat_Jog1PR_trig : Bool;
      stat_Jog2PAux : Bool;
      stat_Jog2PR_trig : Bool;
      stat_Jog1PMode8Aux : Bool;
      stat_Jog1PMode8R_trig : Bool;
      stat_Jog2PMode8Aux : Bool;
      stat_Jog2PMode8R_trig : Bool;
      stat_Status : Word;
      statStartCounter : Int;
      stat_ActMode : Int;
      stat_MaxCounterRetries { ExternalAccessible := 'False'; ExternalVisible := 'False'; ExternalWritable := 'False'} : Int;
   END_VAR

   VAR_TEMP 
      tempDWord : DWord;
      tmpSendBuffer : Array[0..11] of Word;
      tmpReadBuffer : Array[0..11] of Word;
   END_VAR

   VAR CONSTANT 
      MaxCounterStart : Int := 50;
      MAXMODE : Int := 8;
      STATUS_IN_OPERATION : Word := 16#7002;
      ERROR_INVALID_MODE : Word := 16#8202;
      ERROR_OVERRIDE : Word := 16#8203;
      ERROR_INVALID_TRV_BLOCK : Word := 16#8204;
      ERROR_DRIVE_ERROR : Word := 16#8401;
      ERROR_SWITCH_ON_INHIBITED : Word := 16#8402;
      ERROR_DPRD_DAT : Word := 16#8600;
      ERROR_DPWR_DAT : Word := 16#8601;
   END_VAR


BEGIN
	(*############################################################
	    FESTO SE & Co. KG, Esslingen
	    Copyright (c) 2020. All rights reserved.    
	
	    NAME OF FUNCTION BLOCK:         Festo_PTP_Drives_PN
	    VERSION NUMBER:                 V1.5
	    COMPOSER:                       Festo
	    
	    -----------------------------------------------------
	   Date        Name                Activity                                                                              
	   19.03.2020  bkle                created (V1.0)
	   09.03.2021  bkle                name changed
	   18.03.2021  bkle                changed jog behaviour
	   30.07.2021  bkle                Send the StartTask again if ACK is not received - not released
	   06.08.2021  bkle                StartTask is TRUE until ExecuteMode will switch to FALSE
	   22.09.2021  bkle                Added ConfigEpos bits for ReleaseBrake and TravelToFixStop 
	############################################################*)
	
	REGION Check OPM and Override Values
	    // Check the Mode of Operation
	    IF #ModePos > #MAXMODE THEN
	        #Error := True;
	        #stat_Status := #ERROR_INVALID_MODE;
	        #stat_ExecuteIntern := false;
	    ELSIF #ModePos < 1 THEN
	        #Error := True;
	        #stat_Status := #ERROR_INVALID_MODE;
	        #stat_ExecuteIntern := false;
	    ELSE
	        IF #stat_Status = #ERROR_INVALID_MODE THEN
	            #stat_Status := #STATUS_IN_OPERATION;
	            #Error := False;
	        END_IF;
	    END_IF;
	    
	    
	    //Check the Velocity Override 
	    IF (#OverV < 0) OR (#OverV > 199) THEN
	        #stat_Status := #ERROR_OVERRIDE;
	        #Error := True;
	    ELSE
	        // Write Velocity Override into Send Buffer
	        #stat_CycWrite.Override := INT_TO_WORD(REAL_TO_INT(16384.0 * (INT_TO_REAL(#OverV) / 100.0)));
	        IF #stat_Status = #ERROR_OVERRIDE THEN
	            #stat_Status := #STATUS_IN_OPERATION;
	            #Error := False;
	        END_IF;
	    END_IF;
	    
	    //Check the Acceleration Override  (0% - 100%, 100% => W#16#4000)
	    IF (#OverAcc < 0) OR (#OverAcc > 100) THEN
	        #stat_Status := #ERROR_OVERRIDE;
	        #Error := True;
	    ELSE
	        // Write Acceleration Override into Send Buffer
	        #stat_CycWrite.MDI_ACC := INT_TO_WORD(REAL_TO_INT(16384.0 * (INT_TO_REAL(#OverAcc) / 100.0)));
	        IF #stat_Status = #ERROR_OVERRIDE THEN
	            #stat_Status := #STATUS_IN_OPERATION;
	            #Error := False;
	        END_IF;
	    END_IF;
	    
	    //Check the Deceleration Override  (0% - 100%, 100% => W#16#4000)
	    IF (#OverDec < 0) OR (#OverDec > 100) THEN
	        #stat_Status := #ERROR_OVERRIDE;
	        #Error := True;
	    ELSE
	        // Write Deceleration Override into Send Buffer
	        #stat_CycWrite.MDI_DEC := INT_TO_WORD(REAL_TO_INT(16384.0 * (INT_TO_REAL(#OverDec) / 100.0)));
	        IF #stat_Status = #ERROR_OVERRIDE THEN
	            #stat_Status := #STATUS_IN_OPERATION;
	            #Error := False;
	        END_IF;
	    END_IF;
	END_REGION ;
	
	REGION Read Cyclic Data of Telegramm111
	    // Read cyclic telegram 111
	    #stat_RetDPRD := DPRD_DAT(LADDR := #HardwareId,
	                              RECORD => #tmpReadBuffer);
	    
	    //check if the return code is unequal zero -> error occured
	    IF #stat_RetDPRD <> 0 THEN
	        #Error := true;
	        #stat_Status := #ERROR_DPRD_DAT;
	        #DiagID := INT_TO_WORD(#stat_RetDPRD);
	    ELSE
	        
	        // set the Diag status back "in operation"
	        IF #stat_Status = #ERROR_DPRD_DAT THEN
	            #stat_Status := #STATUS_IN_OPERATION;
	            #DiagID := 0;
	            #Error := False;
	        END_IF;
	    END_IF;
	    
	END_REGION ;
	
	
	REGION Read Input from temp data
	    // copy all values from tmp buffer to static data
	    // ZSW1
	    #stat_CycRead.ZSW1.followingErrorInTolerance := #tmpReadBuffer[0].%X8;
	    #stat_CycRead.ZSW1.controlRequest := #tmpReadBuffer[0].%X9;
	    #stat_CycRead.ZSW1.targetPosReached := #tmpReadBuffer[0].%X10;
	    #stat_CycRead.ZSW1.homePosSet := #tmpReadBuffer[0].%X11;
	    #stat_CycRead.ZSW1.acknowledgeTraversingBlockActivated := #tmpReadBuffer[0].%X12;
	    #stat_CycRead.ZSW1.driveStopped := #tmpReadBuffer[0].%X13;
	    #stat_CycRead.ZSW1.axisAccelerates := #tmpReadBuffer[0].%X14;
	    #stat_CycRead.ZSW1.axisDecelerates := #tmpReadBuffer[0].%X15;
	    #stat_CycRead.ZSW1.readyForSwitchOn := #tmpReadBuffer[0].%X0;
	    #stat_CycRead.ZSW1.ready := #tmpReadBuffer[0].%X1;
	    #stat_CycRead.ZSW1.operationEnabled := #tmpReadBuffer[0].%X2;
	    #stat_CycRead.ZSW1.faultPresent := #tmpReadBuffer[0].%X3;
	    #stat_CycRead.ZSW1.noCoastingActive := #tmpReadBuffer[0].%X4;
	    #stat_CycRead.ZSW1.noQuickStopActive := #tmpReadBuffer[0].%X5;
	    #stat_CycRead.ZSW1.switchingOnInhibitedActive := #tmpReadBuffer[0].%X6;
	    #stat_CycRead.ZSW1.warningActive := #tmpReadBuffer[0].%X7;
	    
	    //POS_ZSW1
	    #stat_CycRead.POS_ZSW1 := #tmpReadBuffer[1];
	    #EPosZSW1 := #stat_CycRead.POS_ZSW1;
	    
	    //POS_ZSW2
	    #stat_CycRead.POS_ZSW2 := #tmpReadBuffer[2];
	    #EPosZSW2 := #stat_CycRead.POS_ZSW2;
	    
	    // ZSW2
	    #stat_CycRead.ZSW2.deviceSpecificBit8 := #tmpReadBuffer[3].%X8;
	    #stat_CycRead.ZSW2.deviceSpecificBit9 := #tmpReadBuffer[3].%X9;
	    #stat_CycRead.ZSW2.deviceSpecificBit10 := #tmpReadBuffer[3].%X10;
	    #stat_CycRead.ZSW2.deviceSpecificBit11 := #tmpReadBuffer[3].%X11;
	    #stat_CycRead.ZSW2.doSignOfLifeBit0 := #tmpReadBuffer[3].%X12;
	    #stat_CycRead.ZSW2.doSignOfLifeBit1 := #tmpReadBuffer[3].%X13;
	    #stat_CycRead.ZSW2.doSignOfLifeBit2 := #tmpReadBuffer[3].%X14;
	    #stat_CycRead.ZSW2.doSignOfLifeBit3 := #tmpReadBuffer[3].%X15;
	    #stat_CycRead.ZSW2.deviceSpecificBit0 := #tmpReadBuffer[3].%X0;
	    #stat_CycRead.ZSW2.deviceSpecificBit1 := #tmpReadBuffer[3].%X1;
	    #stat_CycRead.ZSW2.deviceSpecificBit2 := #tmpReadBuffer[3].%X2;
	    #stat_CycRead.ZSW2.deviceSpecificBit3 := #tmpReadBuffer[3].%X3;
	    #stat_CycRead.ZSW2.deviceSpecificBit4 := #tmpReadBuffer[3].%X4;
	    #stat_CycRead.ZSW2.deviceSpecificBit5 := #tmpReadBuffer[3].%X5;
	    #stat_CycRead.ZSW2.deviceSpecificBit6 := #tmpReadBuffer[3].%X6;
	    #stat_CycRead.ZSW2.deviceSpecificBit7 := #tmpReadBuffer[3].%X7;
	    
	    //MELDW
	    #stat_CycRead.MELDW := #tmpReadBuffer[4];
	    
	    //XIST_A
	    #stat_CycRead.XIST_A.%W0 := #tmpReadBuffer[6];
	    #stat_CycRead.XIST_A.%W1 := #tmpReadBuffer[5];
	    
	    //NIST_B
	    #stat_CycRead.NIST_B.%W0 := #tmpReadBuffer[8];
	    #stat_CycRead.NIST_B.%W1 := #tmpReadBuffer[7];
	    
	    //Fault_Code
	    #stat_CycRead.Fault_Code := #tmpReadBuffer[9];
	    
	    //Warn_Code
	    #stat_CycRead.Warn_Code := #tmpReadBuffer[10];
	    
	    //Reserved
	    #stat_CycRead.Reserved := #tmpReadBuffer[11];
	END_REGION ;
	
	// Mapping of the FB Outputs
	#AxisEnabled := #stat_CycRead.ZSW1.operationEnabled;
	#AxisError := #stat_CycRead.ZSW1.faultPresent;
	#AxisWarn := #stat_CycRead.ZSW1.warningActive;
	#AxisPosOk := #stat_CycRead.ZSW1.targetPosReached;
	#AxisRef := #stat_CycRead.ZSW1.homePosSet;
	#AxisAckSetpoint := #stat_CycRead.ZSW1.acknowledgeTraversingBlockActivated;
	#ClampTorqueReached := #stat_CycRead.POS_ZSW2.%X13;
	#AxisSpFixed := #stat_CycRead.ZSW1.driveStopped;
	#ActVelocity := #stat_CycRead.NIST_B;
	
	
	//scaling the ActVelocity output
	IF #BaseSpeedValue <> 0 THEN
	    #ActVelocity := #ActVelocity * ((#BaseSpeedValue / 1073741824.0));
	END_IF;
	
	#ActPosition := #stat_CycRead.XIST_A;
	#ActWarn := #stat_CycRead.Warn_Code;
	#ActFault := #stat_CycRead.Fault_Code;
	#Lockout := #stat_CycRead.ZSW1.switchingOnInhibitedActive;
	
	//Check the drive error and Lockout status
	IF #AxisError THEN
	    #stat_Status := #ERROR_DRIVE_ERROR;
	    #Error := True;
	ELSIF #Lockout THEN
	    #stat_Status := #ERROR_SWITCH_ON_INHIBITED;
	    #Error := True;
	ELSE
	    // error is gone -> set status in operational
	    IF (#stat_Status = #ERROR_DRIVE_ERROR) OR #stat_Status = #ERROR_SWITCH_ON_INHIBITED THEN
	        #stat_Status := #STATUS_IN_OPERATION;
	        #Error := False;
	    END_IF;
	END_IF;
	
	//Enable the Axis
	#stat_CycWrite.STW1.on := #EnableAxis;                       //STW1.0
	
	//fix values for STW1 data
	#stat_CycWrite.STW1.cancelTraversing := #CancelTraversing;   //STW1.4
	#stat_CycWrite.STW1.intermediateStop := #IntermediateStop;   //STW1.5
	#stat_CycWrite.STW1.acknowledgeFault := #AckError;           //STW1.7
	#stat_CycWrite.STW1.controlByPlc := TRUE;                    //STW1.10
	#stat_CycWrite.STW1.enableOperation := TRUE;                 //STW1.3
	
	// copy the position set value into the send struct
	IF #ModePos <> 4 OR #ModePos <> 5 OR #ModePos <> 6 OR #ModePos <> 7 OR #ModePos <> 8 THEN
	    #stat_CycWrite.MDI_TARPOS := #Position;
	ELSE
	    #stat_CycWrite.MDI_TARPOS := 0;
	END_IF;
	
	//copy the velocity set value into the send struct
	#stat_CycWrite.MDI_VELOCITY := #Velocity;
	
	//Jog bits
	// Mode 7
	//Generate the Jog1 Edge
	#stat_Jog1PR_trig := #Jog1 AND NOT #stat_Jog1PAux;
	//Reset the Auxiliary flag 
	#stat_Jog1PAux := #Jog1;
	
	//Generate the Jog2 Edge
	#stat_Jog2PR_trig := #Jog2 AND NOT #stat_Jog2PAux;
	//Reset the Auxiliary flag 
	#stat_Jog2PAux := #Jog2;
	
	//Mode 8
	//Generate the Jog1 Edge
	#stat_Jog1PMode8R_trig := #Jog1 AND NOT #stat_Jog1PMode8Aux;
	//Reset the Auxiliary flag 
	#stat_Jog1PMode8Aux := #Jog1;
	
	//Generate the Jog2 Edge
	#stat_Jog2PMode8R_trig := #Jog2 AND NOT #stat_Jog2PMode8Aux;
	//Reset the Auxiliary flag 
	#stat_Jog2PMode8Aux := #Jog2;
	
	IF #ModePos <> 4 THEN
	    //Start homing
	    #stat_CycWrite.STW1.StartHoming := false;
	END_IF;
	
	//Relative - Absolute
	#stat_CycWrite.POS_STW1.MDI_MOD := false;
	
	//Positive - Negative direction
	#stat_CycWrite.POS_STW1.PosModulo := false;
	#stat_CycWrite.POS_STW1.NegModulo := false;
	
	// setup mode 
	#stat_CycWrite.POS_STW1.SetupMode := false;
	
	// MDI Active
	#stat_CycWrite.POS_STW1.MDI_Activate := false;
	
	//Trackingmode
	#stat_CycWrite.POS_STW2.Trackingmode := false;
	
	//Jog increment
	#stat_CycWrite.POS_STW2.jog_inc := false;
	
	//delete all the record bits
	#stat_CycWrite.POS_STW1.travBlockBit0 := false;
	#stat_CycWrite.POS_STW1.travBlockBit1 := false;
	#stat_CycWrite.POS_STW1.travBlockBit2 := false;
	#stat_CycWrite.POS_STW1.travBlockBit3 := false;
	#stat_CycWrite.POS_STW1.travBlockBit4 := false;
	#stat_CycWrite.POS_STW1.travBlockBit5 := false;
	#stat_CycWrite.POS_STW1.travBlockBit6 := false;
	
	//Check if the drive is ready for a motion
	IF #stat_CycRead.ZSW1.operationEnabled THEN
	    #stat_Ready4Motion := true;
	ELSE
	    #stat_Ready4Motion := false;
	END_IF;
	
	//Generate the Execute Edge for Mode = 4 and 5
	#stat_ExecR_Trig := #ExecuteMode AND NOT #stat_ExecAux;
	//Reset the Auxiliary flag 
	#stat_ExecAux := #ExecuteMode;
	
	// Set the Execute command according to the ModePos
	IF NOT #ExecuteMode THEN
	    #stat_ExecuteIntern := FALSE;
	    #stat_StepHome := 0;
	ELSIF #ExecuteMode AND #stat_Ready4Motion AND NOT (#ModePos = 4 OR #ModePos = 5 OR #ModePos = 7 OR #ModePos = 8) THEN
	    #stat_ExecuteIntern := TRUE;
	    #stat_ActMode := #ModePos;
	    #stat_StepHome := 0;
	ELSIF #stat_ExecR_Trig AND (#ModePos = 4 OR #ModePos = 5) THEN
	    #stat_ActMode := #ModePos;
	    #stat_StepHome := 0;
	ELSIF #ExecuteMode AND (#stat_ActMode = 7 OR #stat_ActMode = 8) THEN
	    #stat_ExecuteIntern := FALSE;
	    #stat_StepHome := 0;
	ELSIF #ExecuteMode AND #ModePos = 4 THEN
	    
	    CASE #stat_StepHome OF
	            
	        0: // homing is active
	            IF NOT #AxisRef THEN
	                #stat_StepHome := 10;
	            ELSIF #AxisError OR (NOT #AxisSpFixed AND #ModePos = 4) THEN
	                #stat_ExecuteIntern := FALSE;
	            END_IF;
	            
	        10: // wait for homing done
	            IF #AxisRef OR #AxisError OR (NOT #stat_Ready4Motion AND #ModePos = 4) OR #ModePos <> #stat_ActMode OR NOT #ExecuteMode THEN
	                #stat_ExecuteIntern := FALSE;
	                #stat_StepHome := 0;
	            END_IF;
	    END_CASE;
	ELSIF #stat_ExecuteIntern AND #ModePos <> #stat_ActMode THEN
	    #stat_ExecuteIntern := false;
	    #stat_StepHome := 0;
	END_IF;
	
	//Reset the jog bits if the ModePos has changed
	IF (#stat_CycWrite.STW1.jog1 OR #stat_CycWrite.STW1.jog2) AND #ModePos <> #stat_ActMode THEN
	    //Set the jog bits to zero
	    #stat_CycWrite.STW1.jog1 := false;
	    #stat_CycWrite.STW1.jog2 := false;
	END_IF;
	
	// Positionig mode with relative movement (MDI)
	IF #ModePos = 1 THEN
	    
	    // Set the MDI bit
	    #stat_CycWrite.POS_STW1.MDI_Activate := true;
	    
	    // positive direction
	    #stat_CycWrite.POS_STW1.PosModulo := #Positive;
	    
	    // #negative direction
	    #stat_CycWrite.POS_STW1.NegModulo := #Negative;
	    
	    // Check if the drive is enabled for a new motion command
	    IF #stat_Ready4Motion THEN
	        
	        IF NOT #stat_CycWrite.STW1.activateTraversing THEN
	            #stat_ExecuteIntern := #stat_ExecR_Trig;
	        END_IF;
	        
	        //Start Traversing Task
	        #stat_CycWrite.STW1.activateTraversing := #stat_ExecuteIntern;
	        
	    END_IF;
	    
	    // Positionig mode with absolute movement (MDI)
	ELSIF #ModePos = 2 THEN
	    
	    // Set the MDI bit
	    #stat_CycWrite.POS_STW1.MDI_Activate := true;
	    
	    //set the Absolute bit
	    #stat_CycWrite.POS_STW1.MDI_MOD := true;
	    
	    // positive direction
	    #stat_CycWrite.POS_STW1.PosModulo := #Positive;
	    
	    // #negative direction
	    #stat_CycWrite.POS_STW1.NegModulo := #Negative;
	    
	    // Check if the drive is enabled for a new motion command
	    IF #stat_Ready4Motion THEN
	        
	        IF NOT #stat_CycWrite.STW1.activateTraversing THEN
	            #stat_ExecuteIntern := #stat_ExecR_Trig;
	        END_IF;
	        
	        //Start Traversing Task
	        #stat_CycWrite.STW1.activateTraversing := #stat_ExecuteIntern;
	        
	    END_IF;
	    
	    // Positioning with setup mode for endless motion
	ELSIF #ModePos = 3 THEN
	    // Set the MDI bit
	    #stat_CycWrite.POS_STW1.MDI_Activate := true;
	    
	    //set the Absolute bit
	    #stat_CycWrite.POS_STW1.MDI_MOD := true;
	    
	    //setup mode
	    #stat_CycWrite.POS_STW1.SetupMode := true;
	    
	    // positive direction
	    #stat_CycWrite.POS_STW1.PosModulo := #Positive;
	    
	    // #negative direction
	    #stat_CycWrite.POS_STW1.NegModulo := #Negative;
	    
	    // Check if the drive is enabled for a new motion command
	    IF #stat_Ready4Motion THEN
	        
	        IF NOT #stat_CycWrite.STW1.activateTraversing THEN
	            #stat_ExecuteIntern := #stat_ExecR_Trig;
	        END_IF;
	        
	        //Start Traversing Task
	        #stat_CycWrite.STW1.activateTraversing := #stat_ExecuteIntern;
	        
	    END_IF;
	    
	    //Homing mode done by the drive due to the parametrized homing method
	ELSIF #ModePos = 4 THEN
	    // positive direction
	    #stat_CycWrite.POS_STW1.PosModulo := #Positive;
	    
	    // #negative direction
	    #stat_CycWrite.POS_STW1.NegModulo := #Negative;
	    
	    // Check if the drive is enabled for a new motion command
	    IF #stat_Ready4Motion THEN
	        
	        //Start homing
	        IF NOT #stat_CycWrite.STW1.StartHoming THEN
	            #stat_ExecuteIntern := #stat_ExecR_Trig;
	        END_IF;
	        
	        #stat_CycWrite.STW1.StartHoming := #stat_ExecuteIntern;
	    END_IF;
	    
	    //set the reference point (actual position)
	ELSIF #ModePos = 5 THEN
	    
	    // check if there is no error in the drive - this function works also when drive is not enabled
	    IF NOT #AxisError THEN
	        
	        //Start homing
	        IF NOT #stat_CycWrite.POS_STW2.SetReferencePoint THEN
	            #stat_ExecuteIntern := #stat_ExecR_Trig;
	        END_IF;
	        //Set the axis zero point
	        #stat_CycWrite.POS_STW2.SetReferencePoint := #stat_ExecuteIntern;
	        
	    END_IF;
	    
	    //Record mode - parametrized records in the drive can be used
	ELSIF #ModePos = 6 THEN
	    
	    //set the position number into the record bits 
	    IF (DINT_TO_INT(#Position) < 0) OR (DINT_TO_INT(#Position) > 127) THEN
	        // Error, wrong record number
	        #stat_Status := #ERROR_INVALID_TRV_BLOCK;
	        #Error := True;
	    ELSE
	        // error is gone -> set status in operational
	        IF #stat_Status = #ERROR_INVALID_TRV_BLOCK THEN
	            #stat_Status := #STATUS_IN_OPERATION;
	            #Error := False;
	        END_IF;
	        
	        // Record bit 0
	        IF (DINT_TO_WORD(#Position) AND W#16#01) = W#16#01 THEN
	            #stat_CycWrite.POS_STW1.travBlockBit0 := true;
	        END_IF;
	        
	        // Record bit 1
	        IF (DINT_TO_WORD(#Position) AND W#16#02) = W#16#02 THEN
	            #stat_CycWrite.POS_STW1.travBlockBit1 := true;
	        END_IF;
	        
	        // Record bit 2
	        IF (DINT_TO_WORD(#Position) AND W#16#04) = W#16#04 THEN
	            #stat_CycWrite.POS_STW1.travBlockBit2 := true;
	        END_IF;
	        
	        // Record bit 3
	        IF (DINT_TO_WORD(#Position) AND W#16#08) = W#16#08 THEN
	            #stat_CycWrite.POS_STW1.travBlockBit3 := true;
	        END_IF;
	        
	        // Record bit 4
	        IF (DINT_TO_WORD(#Position) AND W#16#10) = W#16#10 THEN
	            #stat_CycWrite.POS_STW1.travBlockBit4 := true;
	        END_IF;
	        
	        // Record bit 5
	        IF (DINT_TO_WORD(#Position) AND W#16#20) = W#16#20 THEN
	            #stat_CycWrite.POS_STW1.travBlockBit5 := true;
	        END_IF;
	        
	        // Record bit 6
	        IF (DINT_TO_WORD(#Position) AND W#16#40) = W#16#40 THEN
	            #stat_CycWrite.POS_STW1.travBlockBit6 := true;
	        END_IF;
	        
	        // Check if the drive is enabled for a new motion command
	        IF #stat_Ready4Motion THEN
	            
	            IF NOT #stat_CycWrite.STW1.activateTraversing THEN
	                #stat_ExecuteIntern := #stat_ExecR_Trig;
	            END_IF;
	            
	            //Start Traversing Task
	            #stat_CycWrite.STW1.activateTraversing := #stat_ExecuteIntern;
	            
	        END_IF;
	    END_IF;
	    
	    //Jog mode - positive or negative
	ELSIF #ModePos = 7 THEN
	    
	    // Check if the drive is enabled for a new motion command
	    IF #stat_Ready4Motion THEN
	        
	        IF #stat_Jog1PR_trig AND NOT #Jog2 THEN
	            #stat_CycWrite.STW1.jog1 := TRUE;
	            #stat_ActMode := #ModePos;
	        ELSIF NOT #Jog1 THEN
	            #stat_CycWrite.STW1.jog1 := false;
	        END_IF;
	        
	        IF #stat_Jog2PR_trig AND NOT #Jog1 THEN
	            #stat_CycWrite.STW1.jog2 := TRUE;
	            #stat_ActMode := #ModePos;
	        ELSIF NOT #Jog2 THEN
	            #stat_CycWrite.STW1.jog2 := false;
	        END_IF;
	    ELSE
	        #stat_CycWrite.STW1.jog1 := false;
	        #stat_CycWrite.STW1.jog2 := false;
	        
	    END_IF;
	    
	    // jog incremental mode
	ELSIF #ModePos = 8 THEN
	    
	    // Check if the drive is enabled for a new motion command
	    IF #stat_Ready4Motion THEN
	        
	        //Jog increment
	        #stat_CycWrite.POS_STW2.jog_inc := true;
	        
	        IF #stat_Jog1PMode8R_trig THEN
	            #stat_CycWrite.STW1.jog1 := TRUE;
	            #stat_ActMode := #ModePos;
	        ELSIF NOT #Jog1 THEN
	            #stat_CycWrite.STW1.jog1 := false;
	        END_IF;
	        
	        IF #stat_Jog2PMode8R_trig THEN
	            #stat_CycWrite.STW1.jog2 := TRUE;
	            #stat_ActMode := #ModePos;
	        ELSIF NOT #Jog2 THEN
	            #stat_CycWrite.STW1.jog2 := false;
	        END_IF;
	        
	        IF #stat_Jog1PMode8R_trig AND #stat_Jog2PMode8R_trig THEN
	            #stat_CycWrite.STW1.jog1 := false;
	            #stat_CycWrite.STW1.jog2 := FALSE;
	        END_IF;
	        
	    ELSE
	        #stat_CycWrite.STW1.jog1 := false;
	        #stat_CycWrite.STW1.jog2 := false;
	        
	    END_IF;
	ELSE
	    // modepos < 1 or > 8
	    #stat_ExecuteIntern := false;
	    #stat_CycWrite.STW1.activateTraversing := false;
	    #stat_CycWrite.STW1.StartHoming := false;
	    #stat_CycWrite.POS_STW2.SetReferencePoint := false;
	    #stat_StepHome := 0;
	    #statStartCounter := 0;
	END_IF;
	
	
	REGION ConfigEPos
	    //Maping of the ConfigEPos to the Telegram
	    #stat_CycWrite.STW1.noCoastStop := #ConfigEPos.%X0;         //STW1.1
	    #stat_CycWrite.STW1.noQuickStop := #ConfigEPos.%X1;         //STW1.2
	    #stat_CycWrite.POS_STW2."SW-Limit" := #ConfigEPos.%X2;
	    #stat_CycWrite.POS_STW2."HW-Limit" := #ConfigEPos.%X3;
	    #stat_CycWrite.POS_STW2.ProbeEdgeEval := #ConfigEPos.%X4;
	    #stat_CycWrite.POS_STW2.SelectProbe := #ConfigEPos.%X5;
	    #stat_CycWrite.STW1.ExternalBlockChange := #ConfigEPos.%X6;
	    #stat_CycWrite.POS_STW2.reserved2 := #ConfigEPos.%X7;
	    #stat_CycWrite.POS_STW1.reserved12 := #ConfigEPos.%X8;
	    #stat_CycWrite.STW2.reserved0 := #ConfigEPos.%X9;
	    #stat_CycWrite.STW2.reserved1 := #ConfigEPos.%X10;
	    #stat_CycWrite.STW2.reserved2 := #ConfigEPos.%X11;
	    #stat_CycWrite.STW2.reserved3 := #ConfigEPos.%X12;
	    #stat_CycWrite.STW2.reserved4 := #ConfigEPos.%X13;
	    #stat_CycWrite.STW2.reserved7 := #ConfigEPos.%X14;
	    #stat_CycWrite.STW1.ReleaseBrake := #ReleaseBrake OR #ConfigEPos.%X15;           //STW1.12
	    #stat_CycWrite.STW1.reserved14 := #ConfigEPos.%X16;
	    #stat_CycWrite.STW1.reserved15 := #ConfigEPos.%X17;
	    #stat_CycWrite.POS_STW2.Trackingmode := #ConfigEPos.%X18;    // different mapping to SINA_POS
	    #stat_CycWrite.POS_STW1.reserved7 := #ConfigEPos.%X19;                // reserved
	    #stat_CycWrite.POS_STW1.reserved11 := #ConfigEPos.%X20;               // reserved
	    #stat_CycWrite.POS_STW1.reserved13 := #ConfigEPos.%X21;               // reserved
	    #stat_CycWrite.POS_STW2.reserved13 := #ConfigEPos.%X22;
	    #stat_CycWrite.POS_STW2.reserved4 := #ConfigEPos.%X23;
	    #stat_CycWrite.POS_STW2.reserved6 := #ConfigEPos.%X24;
	    #stat_CycWrite.POS_STW2.reserved7 := #ConfigEPos.%X25;
	    #stat_CycWrite.POS_STW2.reserved12 := #ConfigEPos.%X26;
	    #stat_CycWrite.POS_STW2.reserved13 := #ConfigEPos.%X27;
	    #stat_CycWrite.STW2.reserved5 := #ConfigEPos.%X28;
	    #stat_CycWrite.STW2.reserved6 := #ConfigEPos.%X29;
	    #stat_CycWrite.STW2.TravelToFixStop := #TravelToFixStop OR #ConfigEPos.%X30;     //STW2.8
	    #stat_CycWrite.STW2.reserved9 := #ConfigEPos.%X31;
	END_REGION ;
	
	REGION Write Output to temp data
	    // copy all cyclic data from stat data to tmp buffer
	    ////STW1
	    #tmpSendBuffer[0].%X0 := #stat_CycWrite.STW1.on;
	    #tmpSendBuffer[0].%X1 := #stat_CycWrite.STW1.noCoastStop;
	    #tmpSendBuffer[0].%X2 := #stat_CycWrite.STW1.noQuickStop;
	    #tmpSendBuffer[0].%X3 := #stat_CycWrite.STW1.enableOperation;
	    #tmpSendBuffer[0].%X4 := #stat_CycWrite.STW1.cancelTraversing;
	    #tmpSendBuffer[0].%X5 := #stat_CycWrite.STW1.intermediateStop;
	    #tmpSendBuffer[0].%X6 := #stat_CycWrite.STW1.activateTraversing;
	    #tmpSendBuffer[0].%X7 := #stat_CycWrite.STW1.acknowledgeFault;
	    #tmpSendBuffer[0].%X8 := #stat_CycWrite.STW1.jog1;
	    #tmpSendBuffer[0].%X9 := #stat_CycWrite.STW1.jog2;
	    #tmpSendBuffer[0].%X10 := #stat_CycWrite.STW1.controlByPlc;
	    #tmpSendBuffer[0].%X11 := #stat_CycWrite.STW1.StartHoming;
	    #tmpSendBuffer[0].%X12 := #stat_CycWrite.STW1.ReleaseBrake;
	    #tmpSendBuffer[0].%X13 := #stat_CycWrite.STW1.ExternalBlockChange;
	    #tmpSendBuffer[0].%X14 := #stat_CycWrite.STW1.reserved14;
	    #tmpSendBuffer[0].%X15 := #stat_CycWrite.STW1.reserved15;
	    //POS_STW1
	    #tmpSendBuffer[1].%X0 := #stat_CycWrite.POS_STW1.travBlockBit0;
	    #tmpSendBuffer[1].%X1 := #stat_CycWrite.POS_STW1.travBlockBit1;
	    #tmpSendBuffer[1].%X2 := #stat_CycWrite.POS_STW1.travBlockBit2;
	    #tmpSendBuffer[1].%X3 := #stat_CycWrite.POS_STW1.travBlockBit3;
	    #tmpSendBuffer[1].%X4 := #stat_CycWrite.POS_STW1.travBlockBit4;
	    #tmpSendBuffer[1].%X5 := #stat_CycWrite.POS_STW1.travBlockBit5;
	    #tmpSendBuffer[1].%X6 := #stat_CycWrite.POS_STW1.travBlockBit6;
	    #tmpSendBuffer[1].%X7 := #stat_CycWrite.POS_STW1.reserved7;
	    #tmpSendBuffer[1].%X8 := #stat_CycWrite.POS_STW1.MDI_MOD;
	    #tmpSendBuffer[1].%X9 := #stat_CycWrite.POS_STW1.PosModulo;
	    #tmpSendBuffer[1].%X10 := #stat_CycWrite.POS_STW1.NegModulo;
	    #tmpSendBuffer[1].%X11 := #stat_CycWrite.POS_STW1.reserved11;
	    #tmpSendBuffer[1].%X12 := #stat_CycWrite.POS_STW1.reserved12;
	    #tmpSendBuffer[1].%X13 := #stat_CycWrite.POS_STW1.reserved13;
	    #tmpSendBuffer[1].%X14 := #stat_CycWrite.POS_STW1.SetupMode;
	    #tmpSendBuffer[1].%X15 := #stat_CycWrite.POS_STW1.MDI_Activate;
	    //POS_STW2
	    #tmpSendBuffer[2].%X0 := #stat_CycWrite.POS_STW2.Trackingmode;
	    #tmpSendBuffer[2].%X1 := #stat_CycWrite.POS_STW2.SetReferencePoint;
	    #tmpSendBuffer[2].%X2 := #stat_CycWrite.POS_STW2.reserved2;
	    #tmpSendBuffer[2].%X3 := #stat_CycWrite.POS_STW2.reserved3;
	    #tmpSendBuffer[2].%X4 := #stat_CycWrite.POS_STW2.reserved4;
	    #tmpSendBuffer[2].%X5 := #stat_CycWrite.POS_STW2.jog_inc;
	    #tmpSendBuffer[2].%X6 := #stat_CycWrite.POS_STW2.reserved6;
	    #tmpSendBuffer[2].%X7 := #stat_CycWrite.POS_STW2.reserved7;
	    #tmpSendBuffer[2].%X8 := #stat_CycWrite.POS_STW2.FlyingRef;
	    #tmpSendBuffer[2].%X9 := #stat_CycWrite.POS_STW2.reserved9;
	    #tmpSendBuffer[2].%X10 := #stat_CycWrite.POS_STW2.SelectProbe;
	    #tmpSendBuffer[2].%X11 := #stat_CycWrite.POS_STW2.ProbeEdgeEval;
	    #tmpSendBuffer[2].%X12 := #stat_CycWrite.POS_STW2.reserved12;
	    #tmpSendBuffer[2].%X13 := #stat_CycWrite.POS_STW2.reserved13;
	    #tmpSendBuffer[2].%X14 := #stat_CycWrite.POS_STW2."SW-Limit";
	    #tmpSendBuffer[2].%X15 := #stat_CycWrite.POS_STW2."HW-Limit";
	    //STW2
	    #tmpSendBuffer[3].%X0 := #stat_CycWrite.STW2.reserved0;
	    #tmpSendBuffer[3].%X1 := #stat_CycWrite.STW2.reserved1;
	    #tmpSendBuffer[3].%X2 := #stat_CycWrite.STW2.reserved2;
	    #tmpSendBuffer[3].%X3 := #stat_CycWrite.STW2.reserved3;
	    #tmpSendBuffer[3].%X4 := #stat_CycWrite.STW2.reserved4;
	    #tmpSendBuffer[3].%X5 := #stat_CycWrite.STW2.reserved5;
	    #tmpSendBuffer[3].%X6 := #stat_CycWrite.STW2.reserved6;
	    #tmpSendBuffer[3].%X7 := #stat_CycWrite.STW2.reserved7;
	    #tmpSendBuffer[3].%X8 := #stat_CycWrite.STW2.TravelToFixStop;
	    #tmpSendBuffer[3].%X9 := #stat_CycWrite.STW2.reserved9;
	    #tmpSendBuffer[3].%X10 := #stat_CycWrite.STW2.reserved10;
	    #tmpSendBuffer[3].%X11 := #stat_CycWrite.STW2.reserved11;
	    #tmpSendBuffer[3].%X12 := #stat_CycWrite.STW2.signOfLifeBit0;
	    #tmpSendBuffer[3].%X13 := #stat_CycWrite.STW2.signOfLifeBit1;
	    #tmpSendBuffer[3].%X14 := #stat_CycWrite.STW2.signOfLifeBit2;
	    #tmpSendBuffer[3].%X15 := #stat_CycWrite.STW2.signOfLifeBit3;
	    
	    //Override
	    #tmpSendBuffer[4] := #stat_CycWrite.Override;
	    
	    //TargetPos
	    #tempDWord := DINT_TO_DWORD(#stat_CycWrite.MDI_TARPOS);
	    #tmpSendBuffer[5] := #tempDWord.%W1;
	    #tmpSendBuffer[6] := #tempDWord.%W0;
	    
	    //TargetVelocity
	    #tempDWord := DINT_TO_DWORD(#stat_CycWrite.MDI_VELOCITY);
	    #tmpSendBuffer[7] := #tempDWord.%W1;
	    #tmpSendBuffer[8] := #tempDWord.%W0;
	    
	    // ACC, DEC
	    #tmpSendBuffer[9] := #stat_CycWrite.MDI_ACC;
	    #tmpSendBuffer[10] := #stat_CycWrite.MDI_DEC;
	    #tmpSendBuffer[11] := #stat_CycWrite.reserved11;
	END_REGION ;
	
	REGION Write Cyclic Data of Telegramm 111
	    // Write cyclic telegram 111
	    #stat_RetDPWR := DPWR_DAT(LADDR := #HardwareId,
	                              RECORD := #tmpSendBuffer);
	    
	    // write SETIO status to diagId
	    IF #stat_RetDPWR <> 0 THEN
	        #Error := true;
	        #stat_Status := #ERROR_DPWR_DAT;
	        #DiagID := INT_TO_WORD(#stat_RetDPWR);
	    ELSE
	        // set the Diag status back "in operation"
	        IF #stat_Status = #ERROR_DPWR_DAT THEN
	            #stat_Status := #STATUS_IN_OPERATION;
	            #DiagID := 0;
	            #Error := False;
	        END_IF;
	        
	    END_IF;
	    //Set the Status Output
	    #Status := #stat_Status;
	    #ActMode := #stat_ActMode;
	END_REGION
	
END_FUNCTION_BLOCK

FUNCTION_BLOCK "CMMS_Z1_Movement"   // FB14, LAD
{ S7_Optimized_Access := 'TRUE' }
VERSION : 0.1
   VAR
      FML_REF : "DT_FML_REF";
   END_VAR
   // FML_REF.DeviceType := 'CMMS';
BEGIN

REGION Network 1
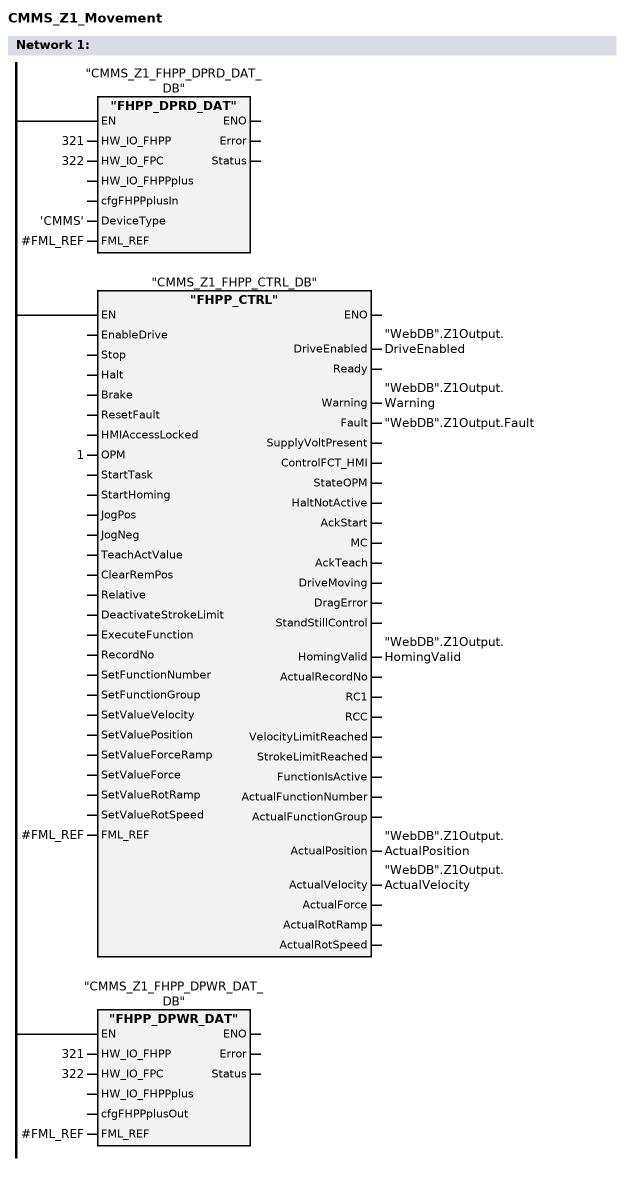
   RUNG wire#powerrail
      "CMMS_Z1_FHPP_DPRD_DAT_DB"(HW_IO_FHPP := 321, HW_IO_FPC := 322, HW_IO_FHPPplus :=, cfgFHPPplusIn :=, DeviceType := 'CMMS', FML_REF := #FML_REF, Error =>, Status =>)
   END_RUNG
   RUNG wire#powerrail
      "CMMS_Z1_FHPP_CTRL_DB"(EnableDrive :=, Stop :=, Halt :=, Brake :=, ResetFault :=, HMIAccessLocked :=, OPM := 1, StartTask :=, StartHoming :=, JogPos :=, JogNeg :=, TeachActValue :=, ClearRemPos :=, Relative :=, DeactivateStrokeLimit :=, ExecuteFunction :=, RecordNo :=, SetFunctionNumber :=, SetFunctionGroup :=, SetValueVelocity :=, SetValuePosition :=, SetValueForceRamp :=, SetValueForce :=, SetValueRotRamp :=, SetValueRotSpeed :=, FML_REF := #FML_REF, DriveEnabled => "WebDB".Z1Output.DriveEnabled, Ready =>, Warning => "WebDB".Z1Output.Warning, Fault => "WebDB".Z1Output.Fault, SupplyVoltPresent =>, ControlFCT_HMI =>, StateOPM =>, HaltNotActive =>, AckStart =>, MC =>, AckTeach =>, DriveMoving =>, DragError =>, StandStillControl =>, HomingValid => "WebDB".Z1Output.HomingValid, ActualRecordNo =>, RC1 =>, RCC =>, VelocityLimitReached =>, StrokeLimitReached =>, FunctionIsActive =>, ActualFunctionNumber =>, ActualFunctionGroup =>, ActualPosition => "WebDB".Z1Output.ActualPosition, ActualVelocity => "WebDB".Z1Output.ActualVelocity, ActualForce =>, ActualRotRamp =>, ActualRotSpeed =>)
   END_RUNG
   RUNG wire#powerrail
      "CMMS_Z1_FHPP_DPWR_DAT_DB"(HW_IO_FHPP := 321, HW_IO_FPC := 322, HW_IO_FHPPplus :=, cfgFHPPplusOut :=, FML_REF := #FML_REF, Error =>, Status =>)
   END_RUNG
   // the same network as SCL:
   "CMMS_Z1_FHPP_DPRD_DAT_DB"(HW_IO_FHPP := 321, HW_IO_FPC := 322, DeviceType := 'CMMS', FML_REF := #FML_REF);   // "FHPP_DPRD_DAT"
   "CMMS_Z1_FHPP_CTRL_DB"(OPM := 1,   // "FHPP_CTRL"
                          FML_REF := #FML_REF,
                          DriveEnabled => "WebDB".Z1Output.DriveEnabled,
                          Warning => "WebDB".Z1Output.Warning,
                          Fault => "WebDB".Z1Output.Fault,
                          HomingValid => "WebDB".Z1Output.HomingValid,
                          ActualPosition => "WebDB".Z1Output.ActualPosition,
                          ActualVelocity => "WebDB".Z1Output.ActualVelocity);
   "CMMS_Z1_FHPP_DPWR_DAT_DB"(HW_IO_FHPP := 321, HW_IO_FPC := 322, FML_REF := #FML_REF);   // "FHPP_DPWR_DAT"
END_REGION
END_FUNCTION_BLOCK

FUNCTION_BLOCK "FHPP_DPRD_DAT"
{ S7_Optimized_Access := 'TRUE' }
AUTHOR : FESTO
FAMILY : 'E-DRIVE'
VERSION : 5.1
   VAR_INPUT 
      HW_IO_FHPP : HW_IO;
      HW_IO_FPC : HW_IO;
   END_VAR
   VAR_INPUT DB_SPECIFIC
      HW_IO_FHPPplus : HW_IO;
      cfgFHPPplusIn : DInt;
   END_VAR
   VAR_INPUT 
      DeviceType : String[16];
   END_VAR

   VAR_OUTPUT 
      Error : Bool;
      Status : "DT_FML_STATUS";
   END_VAR

   VAR_IN_OUT 
      FML_REF : "DT_FML_REF";
   END_VAR

   VAR 
      EnableFHPPplusInOld : DInt;
      FHPPplusSize { ExternalAccessible := 'False'; ExternalVisible := 'False'; ExternalWritable := 'False'} : DInt;
      tmpStatus : "DT_FML_STATUS";
      FHPPplusElementSize { ExternalAccessible := 'False'; ExternalVisible := 'False'; ExternalWritable := 'False'} : Array[1..9] of DInt;
   END_VAR

   VAR_TEMP 
      tmp_bRetVal : Bool;
      FHPPplus8 : Array[1..8] of Byte;
      FHPPplus16 : Array[1..16] of Byte;
      FHPPplus24 : Array[1..24] of Byte;
      WORD_BYTE : Word;
      DWORD_BYTE : DInt;
      i : Int;
      iByteCount : Int;
      tmp_FML_REF : "DT_FML_REF";
   END_VAR


BEGIN
	(*############################################################
	    FESTO AG  Co., Esslingen
	    Copyright (c) 2015. All rights reserved.    
	
	    NAME OF FUNCTION BLOCK:         FHPP_DPRD_DAT
	    VERSION NUMBER:                 V5.1
	    COMPOSER:                       bejk
	    
	    -----------------------------------------------------
	   Date        Name                Activity                                                                              
	   06.08.2015  Benjamin Kilgus     created (V1.0)
	   15.09.2015  Benjamin Kilgus     errorhandling changed (V1.1)
	   14.10.2015  Benjamin Kilgus     check device type added (V1.2)
	   29.08.2016  Benjamin Klein      version changed (V4.1)
	   02.11.2016  Benjamin Klein      adapted to TIAV14 (V5.0)  
	   05.07.2017  Benjamin Klein      optimized function block with Slice access instead of AT (V5.1)
	   18.10.2017  Benjamin Klein      "tmpStatus" at beginning deleted, labels deleted
	############################################################*)
	
	// function block (FB) is busy
	#tmpStatus.Err := FALSE;
	#tmpStatus.Cat := 1;
	#tmpStatus.ID := 16#0000_0002; // FB busy 
	
	// check device type
	IF #DeviceType = 'CMMO_ST' OR
	    #DeviceType = 'EMCA_EC' OR
	    #DeviceType = 'CMMP_AS' OR
	    #DeviceType = 'CMMS_AS' OR
	    #DeviceType = 'CMMS_ST' OR
	    #DeviceType = 'CMMD_AS' THEN
	    
	    #FML_REF.DeviceType := #DeviceType;
	ELSE
	    #tmpStatus.Err := TRUE;
	    #tmpStatus.Cat := 1; // functionblock
	    #tmpStatus.ID := DWORD_TO_DINT(16#8000_001E); // device type not valid
	END_IF;
	
	// ### FHPP Standard ##########################################################
	
	#tmpStatus.ID := DPRD_DAT(LADDR := #HW_IO_FHPP, RECORD => #FML_REF.InData.FHPP);
	
	// #Error WHILE reading?
	IF #tmpStatus.ID <> 0 THEN
	    #tmpStatus.Err := TRUE;
	    #tmpStatus.Cat := 4; // SIEMENS
	END_IF;
	
	// ### FHPP FPC ###############################################################
	IF #HW_IO_FPC <> 0 AND #tmpStatus.Err = FALSE THEN
	    #tmpStatus.ID := INT_TO_WORD(DPRD_DAT(LADDR := #HW_IO_FPC, RECORD => #FML_REF.InData.FPC));
	    
	    // #Error WHILE reading?
	    IF #tmpStatus.ID <> 0 THEN
	        #tmpStatus.Err := TRUE;
	        #tmpStatus.Cat := 4; // SIEMENS
	    END_IF;
	    
	    // mapping of FPC data 
	    #tmp_FML_REF := #FML_REF;
	    #tmp_bRetVal := NOT "FPC_MAPPING"(Mode := FALSE, FML_REF := #tmp_FML_REF);
	    IF #tmp_bRetVal THEN
	        #tmpStatus.Cat := 3; // FPC
	        #tmpStatus.ID := 18;
	    END_IF;
	    #FML_REF := #tmp_FML_REF;
	END_IF;
	
	// ### FHPP PLUS ###############################################################
	IF #HW_IO_FHPPplus <> 0  AND #tmpStatus.Err = FALSE THEN
	    // read FHPPplus data
	    
	    IF #cfgFHPPplusIn <> #EnableFHPPplusInOld THEN
	        #tmpStatus.ID := "FHPPPLUS_MAPPING"(cfgFHPPplus := #cfgFHPPplusIn, FHPPplusElementSize => #FHPPplusElementSize, FHPPplusSize => #FHPPplusSize);
	        #EnableFHPPplusInOld := #cfgFHPPplusIn;
	    END_IF;
	    
	    // FHPP+ Berechnung fehlerhaft beendet
	    IF #tmpStatus.ID <> 0 THEN
	        #tmpStatus.Err := TRUE;
	        #tmpStatus.Cat := 1; // functionblock
	    END_IF;
	    
	    
	    CASE #FHPPplusSize OF
	        0:(* 0 Byte FHPP+ *)
	            (* NO FHPP+ Data configured *)
	            #tmpStatus.Err := TRUE;
	            #tmpStatus.Cat := 1;
	            #tmpStatus.ID := DWORD_TO_DINT(16#8000_0001); // function is called without legal FHPP+ configuration
	            
	        64: // 8 Byte FHPP+ (64bit)
	            #tmpStatus.ID := INT_TO_WORD(DPRD_DAT(LADDR := #HW_IO_FHPPplus, RECORD => #FHPPplus8));
	            IF #tmpStatus.ID <> 0 THEN
	                #tmpStatus.Err := TRUE;
	                #tmpStatus.Cat := 4;
	            END_IF;
	            // copy data to FHPPplus24
	            FOR #i := 1 TO 8 DO
	                #FHPPplus24[#i] := #FHPPplus8[#i];
	            END_FOR;
	            
	        128: // 16 Byte FHPP+ (128bit)        
	            #tmpStatus.ID := INT_TO_WORD(DPRD_DAT(LADDR := #HW_IO_FHPPplus, RECORD => #FHPPplus16));
	            IF #tmpStatus.ID <> 0 THEN
	                #tmpStatus.Err := TRUE;
	                #tmpStatus.Cat := 4;
	            END_IF;
	            // copy data to FHPPplus24
	            FOR #i := 1 TO 16 DO
	                #FHPPplus24[#i] := #FHPPplus16[#i];
	            END_FOR;
	            
	        192: // 24 Byte FHPP+ (192bit)
	            #tmpStatus.ID := INT_TO_WORD(DPRD_DAT(LADDR := #HW_IO_FHPPplus, RECORD => #FHPPplus24));
	            IF #tmpStatus.ID <> 0 THEN
	                #tmpStatus.Err := TRUE;
	                #tmpStatus.Cat := 4;
	            END_IF;
	        ELSE
	            #tmpStatus.Err := TRUE;
	            #tmpStatus.Cat := 1;
	            #tmpStatus.ID := DWORD_TO_DINT(16#8000_0001); //no legal FHPP+ configuration
	    END_CASE;
	    
	    // copy data into FML_REF
	    #iByteCount := 1;
	    FOR #i := 1 TO 9 DO
	        CASE #FHPPplusElementSize[#i] OF
	            0:(* Element is empty *)
	                #FML_REF.InData.FHPPplus[#i] := 0;
	                #iByteCount := #iByteCount + 1;
	            8:(* Element is a BYTE *)
	                #FML_REF.InData.FHPPplus[#i] := #FHPPplus24[#iByteCount];
	                #iByteCount := #iByteCount + 1;
	            16:(* Element is a WORD *)
	                #WORD_BYTE.%B1 := #FHPPplus24[#iByteCount];
	                #WORD_BYTE.%B0 := #FHPPplus24[#iByteCount + 1];
	                #FML_REF.InData.FHPPplus[#i] := #WORD_BYTE;
	                #iByteCount := #iByteCount + 2;
	                
	            32:(* Element is a DWORD *)
	                #DWORD_BYTE.%B3 := #FHPPplus24[#iByteCount];
	                #DWORD_BYTE.%B2 := #FHPPplus24[#iByteCount + 1];
	                #DWORD_BYTE.%B1 := #FHPPplus24[#iByteCount + 2];
	                #DWORD_BYTE.%B0 := #FHPPplus24[#iByteCount + 3];
	                #FML_REF.InData.FHPPplus[#i] := #DWORD_BYTE;
	                #iByteCount := #iByteCount + 4;
	            ELSE
	                #tmpStatus.Err := TRUE;
	                #tmpStatus.Cat := 1;
	                #tmpStatus.ID := DWORD_TO_DINT(16#8000_0001); // //no legal FHPP+ configuration
	        END_CASE;
	    END_FOR;
	END_IF;
	
	// ### EXIT ROUTINE ############################################################
	IF NOT #tmpStatus.Err THEN
	    ENO := TRUE;      // Set ENO-Bit to true
	    #Status := #tmpStatus;
	    #Error := #tmpStatus.Err;
	ELSE
	    ENO := FALSE;     // Set ENO-Bit to false
	    #Status := #tmpStatus;
	    #Error := #tmpStatus.Err;
	END_IF;
END_FUNCTION_BLOCK

FUNCTION "FPC_MAPPING" : Bool
{ S7_Optimized_Access := 'FALSE' }
AUTHOR : FESTO
FAMILY : 'E-DRIVE'
VERSION : 5.1
   VAR_INPUT 
      Mode : Bool;
   END_VAR

   VAR_IN_OUT 
      FML_REF : "DT_FML_REF";
   END_VAR

   VAR_TEMP 
      _Word : Word;
      BByte2 AT _Word : Array[1..2] of Byte;
      _DINT : DInt;
      BByte4 AT _DINT : Array[1..4] of Byte;
      Req_Identifier : Int;
      Resp_Identifier : Int;
   END_VAR

   VAR CONSTANT 
      Const_1 : Byte := 1;
      Const_4 : Byte := 4;
   END_VAR


BEGIN
	(*############################################################
	   FESTO AG  Co., Esslingen
	   Copyright (c) 2015. All rights reserved.    
	
	   NAME OF FUNCTION BLOCK:         FPC_MAPPING
	   VERSION NUMBER:                 V5.1
	   COMPOSER:                       bejk
	   
	-----------------------------------------------------
	   Date        Name                Activity                                                                              
	   06.08.2015  Benjamin Kilgus     created (V1.0)
	   07.07.2017  Benjamin Klein      version changed (V5.1)
	   17.11.2017  Benjamin Klein      resp_identifier enhanced for SFC and MTR
	############################################################*)
	
	(* MAP INPUTS *)
	IF NOT #Mode THEN
	    
	    // Byte1 FPCS            
	    #FML_REF.FPCS_Modus := SHR(IN := (#FML_REF.InData.FPC[1] AND 2#11110000), N := 4);
	    
